// TIA Portal V20 export
FUNCTION_BLOCK "Sequence_1_StackTable"   // FB232, LAD
AUTHOR : ERsystem_FA2_DH. Kim
// stored: IsIECCheckEnabled true, MemoryReserve 100, Namespace Unit1.Em6, SetENOAutomatically false
   VAR
      statSelectedJobNumber { ExternalWritable := 'False'} : DInt;   // Evaluated Job Number
      instSequenceLADStatus { ExternalWritable := 'False'} : "LAF_StatusLadSequence";
      instSequenceLADControl { ExternalWritable := 'False'} : "LAF_ControlLadSequence";
      statTonTime { ExternalAccessible := 'False'; ExternalVisible := 'False'; ExternalWritable := 'False'} : Array[0..3999] of TON_TIME;
   END_VAR
   VAR_TEMP
      tempLoadingDone : Bool;
   END_VAR
   VAR CONSTANT
      delayTime : Time := T#300ms;
      STEP_IDLE : DInt := 1;
      STEP_IMMEDIATE_STOP : DInt := 9001;   // Step executed when an immediate stop command is triggered for the sequence (i.e. when unit is in state aborting)
      JOB_1_STEP_01 : DInt := 101;
      JOB_1_STEP_10 : DInt := 110;
      JOB_1_STEP_11 : DInt := 111;
      JOB_1_STEP_12 : DInt := 112;
      JOB_1_STEP_13 : DInt := 113;
      JOB_1_STEP_20 : DInt := 120;
      JOB_1_STEP_21 : DInt := 121;
      JOB_1_STEP_22 : DInt := 122;
      JOB_1_STEP_30 : DInt := 130;
      JOB_1_STEP_31 : DInt := 131;
      JOB_1_STEP_32 : DInt := 132;
      JOB_1_STEP_40 : DInt := 140;
      JOB_1_STEP_41 : DInt := 141;
      JOB_1_STEP_42 : DInt := 142;
      JOB_1_STEP_50 : DInt := 150;
      JOB_1_STEP_51 : DInt := 151;
      JOB_1_STEP_52 : DInt := 152;
      JOB_1_STEP_60 : DInt := 160;
      JOB_1_STEP_61 : DInt := 161;
      JOB_1_STEP_62 : DInt := 162;
      JOB_1_STEP_70 : DInt := 170;
      JOB_1_STEP_71 : DInt := 171;
      JOB_1_STEP_80 : DInt := 180;
      JOB_1_STEP_81 : DInt := 181;
      JOB_1_STEP_82 : DInt := 182;
      JOB_1_STEP_83 : DInt := 183;
      JOB_1_STEP_84 : DInt := 184;
      JOB_1_STEP_85 : DInt := 185;
      JOB_1_STEP_90 : DInt := 190;
      JOB_2_STEP_01 : DInt := 201;
      JOB_2_STEP_10 : DInt := 210;
      JOB_2_STEP_20 : DInt := 220;
      JOB_2_STEP_80 : DInt := 280;
      JOB_2_STEP_90 : DInt := 290;
      JOB_12_STEP_01 : DInt := 1201;
      JOB_12_STEP_10 : DInt := 1210;
      JOB_12_STEP_90 : DInt := 1290;
      JOB_13_STEP_01 : DInt := 1301;
      JOB_13_STEP_10 : DInt := 1310;
      JOB_13_STEP_90 : DInt := 1390;
      JOB_4_STEP_01 : DInt := 401;
      JOB_4_STEP_10 : DInt := 410;
      JOB_4_STEP_20 : DInt := 420;
      JOB_4_STEP_21 : DInt := 421;
      JOB_4_STEP_30 : DInt := 430;
      JOB_4_STEP_31 : DInt := 431;
      JOB_4_STEP_40 : DInt := 440;
      JOB_4_STEP_41 : DInt := 441;
      JOB_4_STEP_50 : DInt := 450;
      JOB_4_STEP_80 : DInt := 480;
      JOB_4_STEP_90 : DInt := 490;
      JOB_22_STEP_01 : DInt := 2201;
      JOB_22_STEP_10 : DInt := 2210;
      JOB_22_STEP_20 : DInt := 2220;
      JOB_22_STEP_21 : DInt := 2221;
      JOB_22_STEP_22 : DInt := 2222;
      JOB_22_STEP_80 : DInt := 2280;
      JOB_22_STEP_90 : DInt := 2290;
      JOB_23_STEP_01 : DInt := 2301;
      JOB_23_STEP_10 : DInt := 2310;
      JOB_23_STEP_20 : DInt := 2320;
      JOB_23_STEP_21 : DInt := 2321;
      JOB_23_STEP_22 : DInt := 2322;
      JOB_23_STEP_80 : DInt := 2380;
      JOB_23_STEP_90 : DInt := 2390;
      JOB_30_STEP_01 : DInt := 3001;
      JOB_30_STEP_10 : DInt := 3010;
      JOB_30_STEP_20 : DInt := 3020;
      JOB_30_STEP_90 : DInt := 3090;
      JOB_31_STEP_01 : DInt := 3101;
      JOB_31_STEP_10 : DInt := 3110;
      JOB_31_STEP_90 : DInt := 3190;
      FALSE : Bool := FALSE;
      TRUE : Bool := TRUE;
   END_VAR
   VAR_TEMP   // added for the SCL form of the ladder/FBD networks
      _w1 : Bool;
   END_VAR
BEGIN

REGION Network 1: BLOCK INFO HEADER
   // (company) / (C) Copyright (year)
   // ---------------------------------------------------------------------------------
   // Title:                             (Title of this block)
   // Comment/Function: (that is implemented in the block)
   // Library/Family:           (that the source is dedicated to)
   // Author:                        (department / person in charge / contact)
   // Target System:          (test system with FW version)
   // Engineering:              TIA Portal (SW version)
   // Restrictions:               (OB types, etc.)
   // Requirements:           (hardware, technological package, etc.)
   // ---------------------------------------------------------------------------------
   // Change log table:
   // Version          | Date             | Signature      | Expert in charge  | Changes applied ------------------------|----------------------|-------------------------|--------------------------------|-----------------------
   // 001.000.000 | yyyy-mm-dd | 0x00000000 | (name of expert) | First released version
END_REGION

REGION Network 2: DESCRIPTION
   // This is a template block provided by the Automation Framework. It can be used to create an own project.
   // The Block Info Header is prepared to put in your own data.
   // Description of the block could be added here and the docu created by Code2Docu.
END_REGION

REGION Network 3: ********************* CONTROL *************************
END_REGION

REGION Network 4: Sequence Control
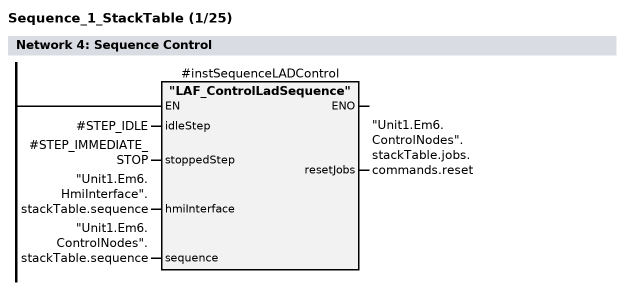
   RUNG wire#powerrail
      #instSequenceLADControl(idleStep := #STEP_IDLE, stoppedStep := #STEP_IMMEDIATE_STOP, hmiInterface := "Unit1.Em6.HmiInterface".stackTable.sequence, sequence := "Unit1.Em6.ControlNodes".stackTable.sequence, resetJobs => "Unit1.Em6.ControlNodes".stackTable.jobs.commands.reset)
   END_RUNG
   // the same network as SCL:
   #instSequenceLADControl(idleStep := #STEP_IDLE,   // "LAF_ControlLadSequence"
                           stoppedStep := #STEP_IMMEDIATE_STOP,
                           hmiInterface := "Unit1.Em6.HmiInterface".stackTable.sequence,
                           sequence := "Unit1.Em6.ControlNodes".stackTable.sequence,
                           resetJobs => "Unit1.Em6.ControlNodes".stackTable.jobs.commands.reset);
END_REGION

REGION Network 5: *************** JOB SELECT **************************
END_REGION

REGION Network 6: STEP IDLE
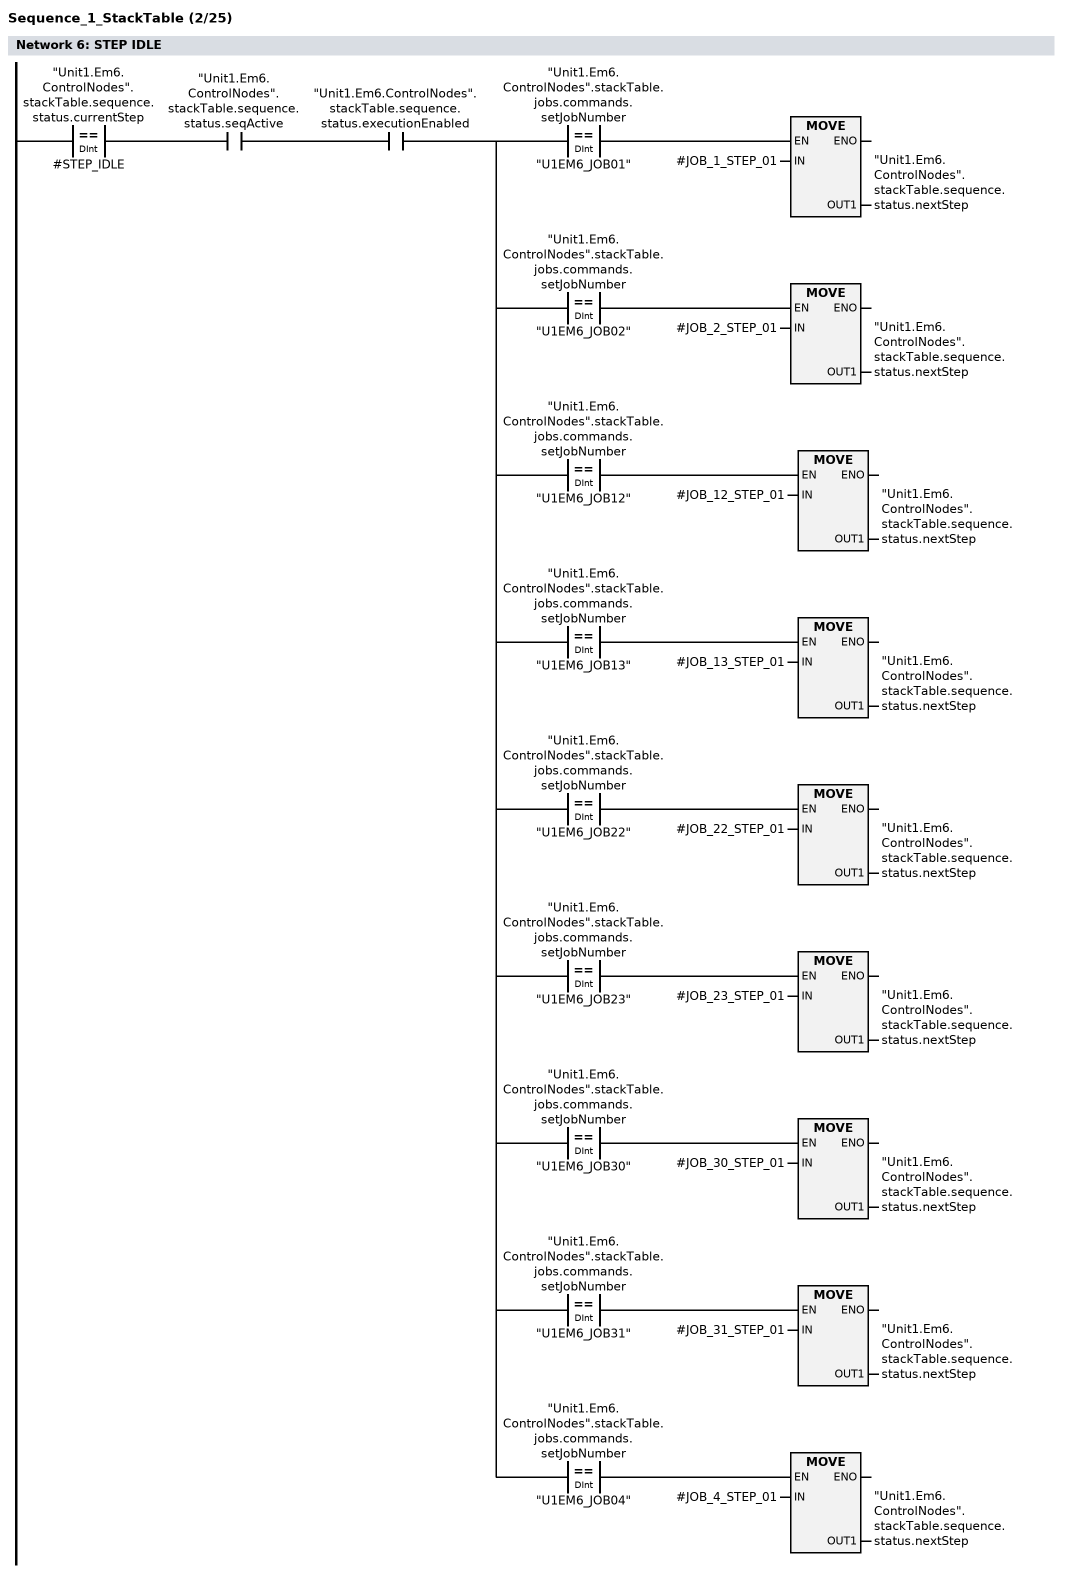
   RUNG wire#powerrail
      { S7_Templates := "SrcType := DInt" } EQ_Contact(in1 := "Unit1.Em6.ControlNodes".stackTable.sequence.status.currentStep, in2 := #STEP_IDLE)
      Contact( "Unit1.Em6.ControlNodes".stackTable.sequence.status.seqActive )
      Contact( "Unit1.Em6.ControlNodes".stackTable.sequence.status.executionEnabled )
      wire#w1
      { S7_Templates := "SrcType := DInt" } EQ_Contact(in1 := "Unit1.Em6.ControlNodes".stackTable.jobs.commands.setJobNumber, in2 := "U1EM6_JOB01")
      Move(in := #JOB_1_STEP_01, out1 => "Unit1.Em6.ControlNodes".stackTable.sequence.status.nextStep)
   END_RUNG
   RUNG wire#w1
      { S7_Templates := "SrcType := DInt" } EQ_Contact(in1 := "Unit1.Em6.ControlNodes".stackTable.jobs.commands.setJobNumber, in2 := "U1EM6_JOB02")
      Move(in := #JOB_2_STEP_01, out1 => "Unit1.Em6.ControlNodes".stackTable.sequence.status.nextStep)
   END_RUNG
   RUNG wire#w1
      { S7_Templates := "SrcType := DInt" } EQ_Contact(in1 := "Unit1.Em6.ControlNodes".stackTable.jobs.commands.setJobNumber, in2 := "U1EM6_JOB12")
      Move(in := #JOB_12_STEP_01, out1 => "Unit1.Em6.ControlNodes".stackTable.sequence.status.nextStep)
   END_RUNG
   RUNG wire#w1
      { S7_Templates := "SrcType := DInt" } EQ_Contact(in1 := "Unit1.Em6.ControlNodes".stackTable.jobs.commands.setJobNumber, in2 := "U1EM6_JOB13")
      Move(in := #JOB_13_STEP_01, out1 => "Unit1.Em6.ControlNodes".stackTable.sequence.status.nextStep)
   END_RUNG
   RUNG wire#w1
      { S7_Templates := "SrcType := DInt" } EQ_Contact(in1 := "Unit1.Em6.ControlNodes".stackTable.jobs.commands.setJobNumber, in2 := "U1EM6_JOB22")
      Move(in := #JOB_22_STEP_01, out1 => "Unit1.Em6.ControlNodes".stackTable.sequence.status.nextStep)
   END_RUNG
   RUNG wire#w1
      { S7_Templates := "SrcType := DInt" } EQ_Contact(in1 := "Unit1.Em6.ControlNodes".stackTable.jobs.commands.setJobNumber, in2 := "U1EM6_JOB23")
      Move(in := #JOB_23_STEP_01, out1 => "Unit1.Em6.ControlNodes".stackTable.sequence.status.nextStep)
   END_RUNG
   RUNG wire#w1
      { S7_Templates := "SrcType := DInt" } EQ_Contact(in1 := "Unit1.Em6.ControlNodes".stackTable.jobs.commands.setJobNumber, in2 := "U1EM6_JOB30")
      Move(in := #JOB_30_STEP_01, out1 => "Unit1.Em6.ControlNodes".stackTable.sequence.status.nextStep)
   END_RUNG
   RUNG wire#w1
      { S7_Templates := "SrcType := DInt" } EQ_Contact(in1 := "Unit1.Em6.ControlNodes".stackTable.jobs.commands.setJobNumber, in2 := "U1EM6_JOB31")
      Move(in := #JOB_31_STEP_01, out1 => "Unit1.Em6.ControlNodes".stackTable.sequence.status.nextStep)
   END_RUNG
   RUNG wire#w1
      { S7_Templates := "SrcType := DInt" } EQ_Contact(in1 := "Unit1.Em6.ControlNodes".stackTable.jobs.commands.setJobNumber, in2 := "U1EM6_JOB04")
      Move(in := #JOB_4_STEP_01, out1 => "Unit1.Em6.ControlNodes".stackTable.sequence.status.nextStep)
   END_RUNG
   // the same network as SCL:
   #_w1 := ("Unit1.Em6.ControlNodes".stackTable.sequence.status.currentStep = #STEP_IDLE) AND "Unit1.Em6.ControlNodes".stackTable.sequence.status.seqActive AND "Unit1.Em6.ControlNodes".stackTable.sequence.status.executionEnabled;
   IF #_w1 AND ("Unit1.Em6.ControlNodes".stackTable.jobs.commands.setJobNumber = "U1EM6_JOB01") THEN
       "Unit1.Em6.ControlNodes".stackTable.sequence.status.nextStep := #JOB_1_STEP_01;
   END_IF;
   IF #_w1 AND ("Unit1.Em6.ControlNodes".stackTable.jobs.commands.setJobNumber = "U1EM6_JOB02") THEN
       "Unit1.Em6.ControlNodes".stackTable.sequence.status.nextStep := #JOB_2_STEP_01;
   END_IF;
   IF #_w1 AND ("Unit1.Em6.ControlNodes".stackTable.jobs.commands.setJobNumber = "U1EM6_JOB12") THEN
       "Unit1.Em6.ControlNodes".stackTable.sequence.status.nextStep := #JOB_12_STEP_01;
   END_IF;
   IF #_w1 AND ("Unit1.Em6.ControlNodes".stackTable.jobs.commands.setJobNumber = "U1EM6_JOB13") THEN
       "Unit1.Em6.ControlNodes".stackTable.sequence.status.nextStep := #JOB_13_STEP_01;
   END_IF;
   IF #_w1 AND ("Unit1.Em6.ControlNodes".stackTable.jobs.commands.setJobNumber = "U1EM6_JOB22") THEN
       "Unit1.Em6.ControlNodes".stackTable.sequence.status.nextStep := #JOB_22_STEP_01;
   END_IF;
   IF #_w1 AND ("Unit1.Em6.ControlNodes".stackTable.jobs.commands.setJobNumber = "U1EM6_JOB23") THEN
       "Unit1.Em6.ControlNodes".stackTable.sequence.status.nextStep := #JOB_23_STEP_01;
   END_IF;
   IF #_w1 AND ("Unit1.Em6.ControlNodes".stackTable.jobs.commands.setJobNumber = "U1EM6_JOB30") THEN
       "Unit1.Em6.ControlNodes".stackTable.sequence.status.nextStep := #JOB_30_STEP_01;
   END_IF;
   IF #_w1 AND ("Unit1.Em6.ControlNodes".stackTable.jobs.commands.setJobNumber = "U1EM6_JOB31") THEN
       "Unit1.Em6.ControlNodes".stackTable.sequence.status.nextStep := #JOB_31_STEP_01;
   END_IF;
   IF #_w1 AND ("Unit1.Em6.ControlNodes".stackTable.jobs.commands.setJobNumber = "U1EM6_JOB04") THEN
       "Unit1.Em6.ControlNodes".stackTable.sequence.status.nextStep := #JOB_4_STEP_01;
   END_IF;
END_REGION

REGION Network 7: *************** JOB[1] EM HOMING ************************
END_REGION

REGION Network 8: Step[101] : JOB[1] Condition
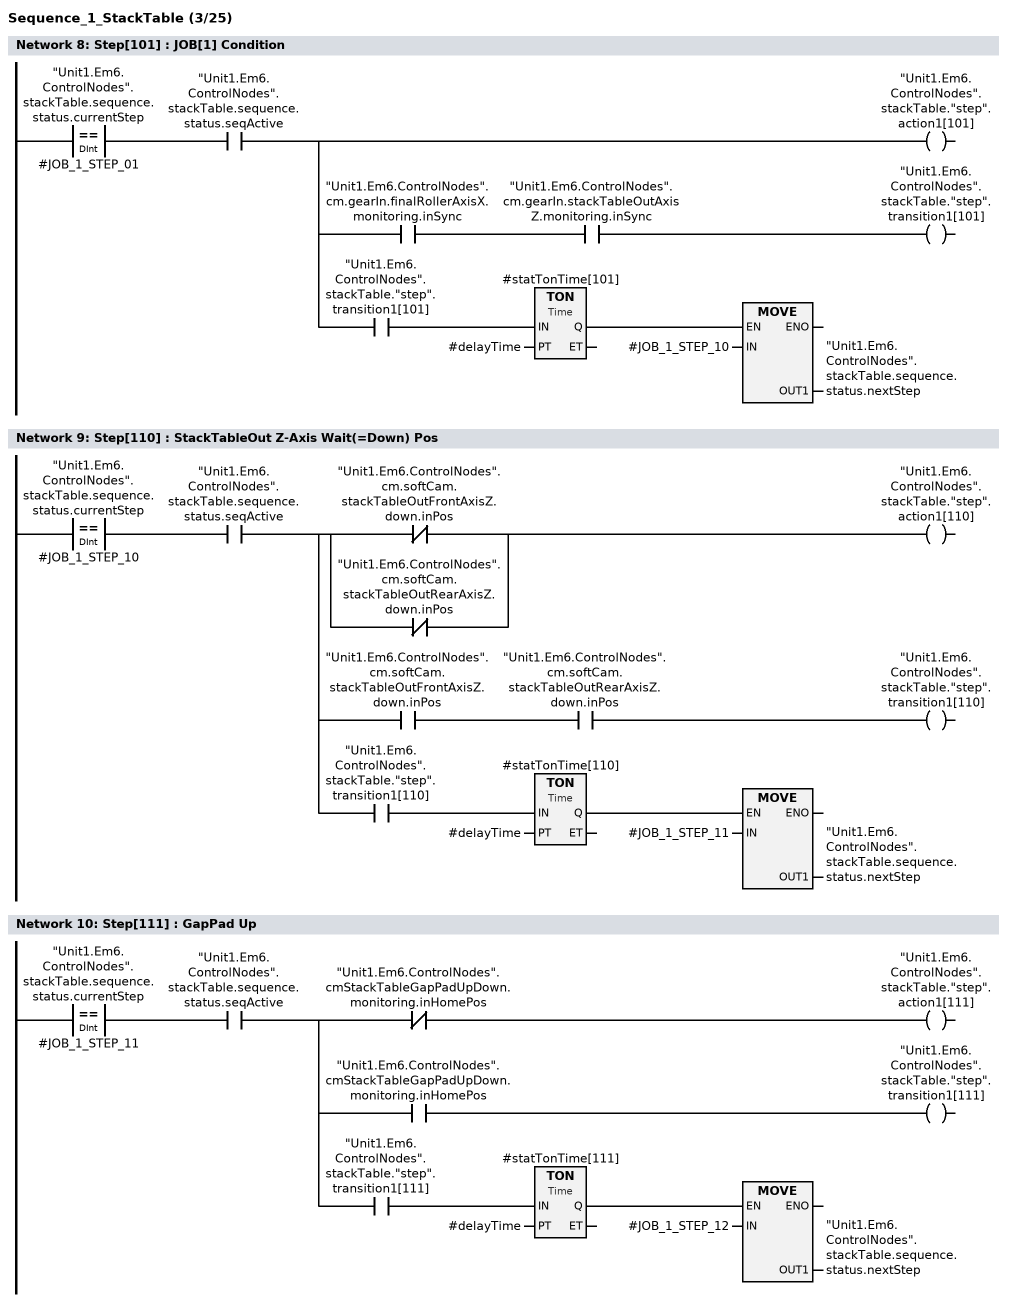
   RUNG wire#powerrail
      { S7_Templates := "SrcType := DInt" } EQ_Contact(in1 := "Unit1.Em6.ControlNodes".stackTable.sequence.status.currentStep, in2 := #JOB_1_STEP_01)
      Contact( "Unit1.Em6.ControlNodes".stackTable.sequence.status.seqActive )
      wire#w1
      Coil( "Unit1.Em6.ControlNodes".stackTable."step".action1[101] )
   END_RUNG
   RUNG wire#w1
      Contact( "Unit1.Em6.ControlNodes".cm.gearIn.finalRollerAxisX.monitoring.inSync )
      Contact( "Unit1.Em6.ControlNodes".cm.gearIn.stackTableOutAxisZ.monitoring.inSync )
      Coil( "Unit1.Em6.ControlNodes".stackTable."step".transition1[101] )
   END_RUNG
   RUNG wire#w1
      Contact( "Unit1.Em6.ControlNodes".stackTable."step".transition1[101] )
      { S7_Templates := "time_type := Time" } #statTonTime[101].TON(pt := #delayTime, et =>)
      Move(in := #JOB_1_STEP_10, out1 => "Unit1.Em6.ControlNodes".stackTable.sequence.status.nextStep)
   END_RUNG
   // the same network as SCL:
   "Unit1.Em6.ControlNodes".stackTable."step".action1[101] := ("Unit1.Em6.ControlNodes".stackTable.sequence.status.currentStep = #JOB_1_STEP_01) AND "Unit1.Em6.ControlNodes".stackTable.sequence.status.seqActive;
   "Unit1.Em6.ControlNodes".stackTable."step".transition1[101] := ("Unit1.Em6.ControlNodes".stackTable.sequence.status.currentStep = #JOB_1_STEP_01) AND "Unit1.Em6.ControlNodes".stackTable.sequence.status.seqActive AND "Unit1.Em6.ControlNodes".cm.gearIn.finalRollerAxisX.monitoring.inSync AND "Unit1.Em6.ControlNodes".cm.gearIn.stackTableOutAxisZ.monitoring.inSync;
   #statTonTime[101].TON(IN := ("Unit1.Em6.ControlNodes".stackTable.sequence.status.currentStep = #JOB_1_STEP_01) AND "Unit1.Em6.ControlNodes".stackTable.sequence.status.seqActive AND "Unit1.Em6.ControlNodes".stackTable."step".transition1[101],
                         PT := #delayTime);
   IF #statTonTime[101].Q THEN
       "Unit1.Em6.ControlNodes".stackTable.sequence.status.nextStep := #JOB_1_STEP_10;
   END_IF;
END_REGION

REGION Network 9: Step[110] : StackTableOut Z-Axis Wait(=Down) Pos
   RUNG wire#powerrail
      { S7_Templates := "SrcType := DInt" } EQ_Contact(in1 := "Unit1.Em6.ControlNodes".stackTable.sequence.status.currentStep, in2 := #JOB_1_STEP_10)
      Contact( "Unit1.Em6.ControlNodes".stackTable.sequence.status.seqActive )
      wire#w1
      I_Contact( "Unit1.Em6.ControlNodes".cm.softCam.stackTableOutFrontAxisZ.down.inPos )
      wire#w2
      Coil( "Unit1.Em6.ControlNodes".stackTable."step".action1[110] )
   END_RUNG
   RUNG wire#w1
      I_Contact( "Unit1.Em6.ControlNodes".cm.softCam.stackTableOutRearAxisZ.down.inPos )
   END_RUNG wire#w2
   RUNG wire#w1
      Contact( "Unit1.Em6.ControlNodes".cm.softCam.stackTableOutFrontAxisZ.down.inPos )
      Contact( "Unit1.Em6.ControlNodes".cm.softCam.stackTableOutRearAxisZ.down.inPos )
      Coil( "Unit1.Em6.ControlNodes".stackTable."step".transition1[110] )
   END_RUNG
   RUNG wire#w1
      Contact( "Unit1.Em6.ControlNodes".stackTable."step".transition1[110] )
      { S7_Templates := "time_type := Time" } #statTonTime[110].TON(pt := #delayTime, et =>)
      Move(in := #JOB_1_STEP_11, out1 => "Unit1.Em6.ControlNodes".stackTable.sequence.status.nextStep)
   END_RUNG
   // the same network as SCL:
   #_w1 := ("Unit1.Em6.ControlNodes".stackTable.sequence.status.currentStep = #JOB_1_STEP_10) AND "Unit1.Em6.ControlNodes".stackTable.sequence.status.seqActive;
   "Unit1.Em6.ControlNodes".stackTable."step".action1[110] := #_w1 AND (NOT "Unit1.Em6.ControlNodes".cm.softCam.stackTableOutFrontAxisZ.down.inPos OR NOT "Unit1.Em6.ControlNodes".cm.softCam.stackTableOutRearAxisZ.down.inPos);
   "Unit1.Em6.ControlNodes".stackTable."step".transition1[110] := #_w1 AND "Unit1.Em6.ControlNodes".cm.softCam.stackTableOutFrontAxisZ.down.inPos AND "Unit1.Em6.ControlNodes".cm.softCam.stackTableOutRearAxisZ.down.inPos;
   #statTonTime[110].TON(IN := #_w1 AND "Unit1.Em6.ControlNodes".stackTable."step".transition1[110],
                         PT := #delayTime);
   IF #statTonTime[110].Q THEN
       "Unit1.Em6.ControlNodes".stackTable.sequence.status.nextStep := #JOB_1_STEP_11;
   END_IF;
END_REGION

REGION Network 10: Step[111] : GapPad Up
   RUNG wire#powerrail
      { S7_Templates := "SrcType := DInt" } EQ_Contact(in1 := "Unit1.Em6.ControlNodes".stackTable.sequence.status.currentStep, in2 := #JOB_1_STEP_11)
      Contact( "Unit1.Em6.ControlNodes".stackTable.sequence.status.seqActive )
      wire#w1
      I_Contact( "Unit1.Em6.ControlNodes".cmStackTableGapPadUpDown.monitoring.inHomePos )
      Coil( "Unit1.Em6.ControlNodes".stackTable."step".action1[111] )
   END_RUNG
   RUNG wire#w1
      Contact( "Unit1.Em6.ControlNodes".cmStackTableGapPadUpDown.monitoring.inHomePos )
      Coil( "Unit1.Em6.ControlNodes".stackTable."step".transition1[111] )
   END_RUNG
   RUNG wire#w1
      Contact( "Unit1.Em6.ControlNodes".stackTable."step".transition1[111] )
      { S7_Templates := "time_type := Time" } #statTonTime[111].TON(pt := #delayTime, et =>)
      Move(in := #JOB_1_STEP_12, out1 => "Unit1.Em6.ControlNodes".stackTable.sequence.status.nextStep)
   END_RUNG
   // the same network as SCL:
   #_w1 := ("Unit1.Em6.ControlNodes".stackTable.sequence.status.currentStep = #JOB_1_STEP_11) AND "Unit1.Em6.ControlNodes".stackTable.sequence.status.seqActive;
   "Unit1.Em6.ControlNodes".stackTable."step".action1[111] := #_w1 AND NOT "Unit1.Em6.ControlNodes".cmStackTableGapPadUpDown.monitoring.inHomePos;
   "Unit1.Em6.ControlNodes".stackTable."step".transition1[111] := #_w1 AND "Unit1.Em6.ControlNodes".cmStackTableGapPadUpDown.monitoring.inHomePos;
   #statTonTime[111].TON(IN := #_w1 AND "Unit1.Em6.ControlNodes".stackTable."step".transition1[111],
                         PT := #delayTime);
   IF #statTonTime[111].Q THEN
       "Unit1.Em6.ControlNodes".stackTable.sequence.status.nextStep := #JOB_1_STEP_12;
   END_IF;
END_REGION

REGION Network 11: Step[112] : A,C.Mendrel Clamp Work Pos
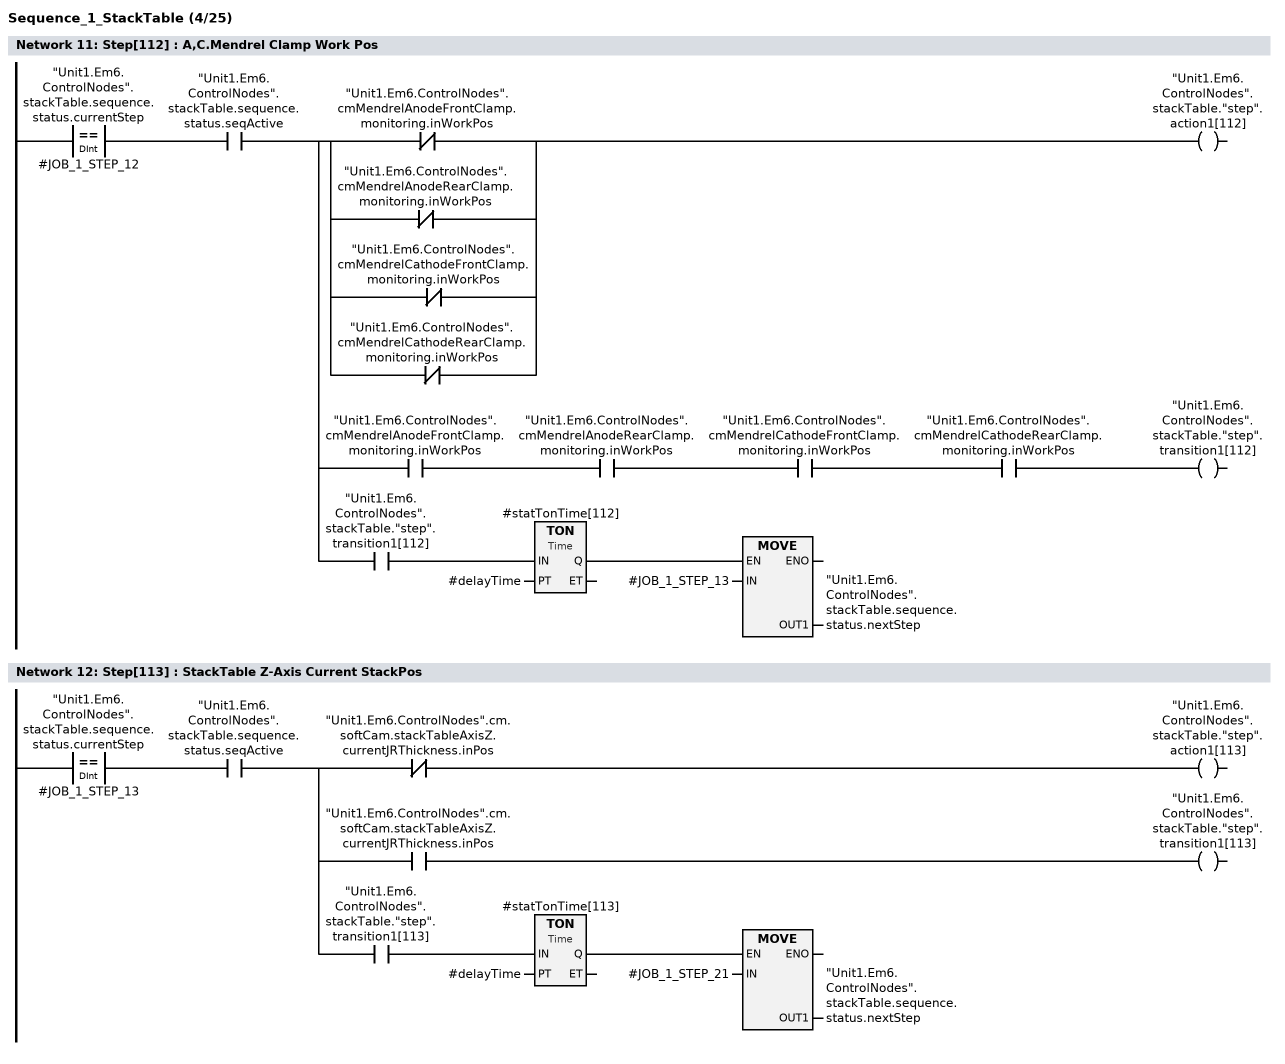
   RUNG wire#powerrail
      { S7_Templates := "SrcType := DInt" } EQ_Contact(in1 := "Unit1.Em6.ControlNodes".stackTable.sequence.status.currentStep, in2 := #JOB_1_STEP_12)
      Contact( "Unit1.Em6.ControlNodes".stackTable.sequence.status.seqActive )
      wire#w1
      I_Contact( "Unit1.Em6.ControlNodes".cmMendrelAnodeFrontClamp.monitoring.inWorkPos )
      wire#w2
      Coil( "Unit1.Em6.ControlNodes".stackTable."step".action1[112] )
   END_RUNG
   RUNG wire#w1
      I_Contact( "Unit1.Em6.ControlNodes".cmMendrelAnodeRearClamp.monitoring.inWorkPos )
   END_RUNG wire#w2
   RUNG wire#w1
      I_Contact( "Unit1.Em6.ControlNodes".cmMendrelCathodeFrontClamp.monitoring.inWorkPos )
   END_RUNG wire#w2
   RUNG wire#w1
      I_Contact( "Unit1.Em6.ControlNodes".cmMendrelCathodeRearClamp.monitoring.inWorkPos )
   END_RUNG wire#w2
   RUNG wire#w1
      Contact( "Unit1.Em6.ControlNodes".cmMendrelAnodeFrontClamp.monitoring.inWorkPos )
      Contact( "Unit1.Em6.ControlNodes".cmMendrelAnodeRearClamp.monitoring.inWorkPos )
      Contact( "Unit1.Em6.ControlNodes".cmMendrelCathodeFrontClamp.monitoring.inWorkPos )
      Contact( "Unit1.Em6.ControlNodes".cmMendrelCathodeRearClamp.monitoring.inWorkPos )
      Coil( "Unit1.Em6.ControlNodes".stackTable."step".transition1[112] )
   END_RUNG
   RUNG wire#w1
      Contact( "Unit1.Em6.ControlNodes".stackTable."step".transition1[112] )
      { S7_Templates := "time_type := Time" } #statTonTime[112].TON(pt := #delayTime, et =>)
      Move(in := #JOB_1_STEP_13, out1 => "Unit1.Em6.ControlNodes".stackTable.sequence.status.nextStep)
   END_RUNG
   // the same network as SCL:
   #_w1 := ("Unit1.Em6.ControlNodes".stackTable.sequence.status.currentStep = #JOB_1_STEP_12) AND "Unit1.Em6.ControlNodes".stackTable.sequence.status.seqActive;
   "Unit1.Em6.ControlNodes".stackTable."step".action1[112] := #_w1 AND (NOT "Unit1.Em6.ControlNodes".cmMendrelAnodeFrontClamp.monitoring.inWorkPos OR NOT "Unit1.Em6.ControlNodes".cmMendrelAnodeRearClamp.monitoring.inWorkPos OR NOT "Unit1.Em6.ControlNodes".cmMendrelCathodeFrontClamp.monitoring.inWorkPos OR NOT "Unit1.Em6.ControlNodes".cmMendrelCathodeRearClamp.monitoring.inWorkPos);
   "Unit1.Em6.ControlNodes".stackTable."step".transition1[112] := #_w1 AND "Unit1.Em6.ControlNodes".cmMendrelAnodeFrontClamp.monitoring.inWorkPos AND "Unit1.Em6.ControlNodes".cmMendrelAnodeRearClamp.monitoring.inWorkPos AND "Unit1.Em6.ControlNodes".cmMendrelCathodeFrontClamp.monitoring.inWorkPos AND "Unit1.Em6.ControlNodes".cmMendrelCathodeRearClamp.monitoring.inWorkPos;
   #statTonTime[112].TON(IN := #_w1 AND "Unit1.Em6.ControlNodes".stackTable."step".transition1[112],
                         PT := #delayTime);
   IF #statTonTime[112].Q THEN
       "Unit1.Em6.ControlNodes".stackTable.sequence.status.nextStep := #JOB_1_STEP_13;
   END_IF;
END_REGION

REGION Network 12: Step[113] : StackTable Z-Axis Current StackPos
   RUNG wire#powerrail
      { S7_Templates := "SrcType := DInt" } EQ_Contact(in1 := "Unit1.Em6.ControlNodes".stackTable.sequence.status.currentStep, in2 := #JOB_1_STEP_13)
      Contact( "Unit1.Em6.ControlNodes".stackTable.sequence.status.seqActive )
      wire#w1
      I_Contact( "Unit1.Em6.ControlNodes".cm.softCam.stackTableAxisZ.currentJRThickness.inPos )
      Coil( "Unit1.Em6.ControlNodes".stackTable."step".action1[113] )
   END_RUNG
   RUNG wire#w1
      Contact( "Unit1.Em6.ControlNodes".cm.softCam.stackTableAxisZ.currentJRThickness.inPos )
      Coil( "Unit1.Em6.ControlNodes".stackTable."step".transition1[113] )
   END_RUNG
   RUNG wire#w1
      Contact( "Unit1.Em6.ControlNodes".stackTable."step".transition1[113] )
      { S7_Templates := "time_type := Time" } #statTonTime[113].TON(pt := #delayTime, et =>)
      Move(in := #JOB_1_STEP_21, out1 => "Unit1.Em6.ControlNodes".stackTable.sequence.status.nextStep)
   END_RUNG
   // the same network as SCL:
   #_w1 := ("Unit1.Em6.ControlNodes".stackTable.sequence.status.currentStep = #JOB_1_STEP_13) AND "Unit1.Em6.ControlNodes".stackTable.sequence.status.seqActive;
   "Unit1.Em6.ControlNodes".stackTable."step".action1[113] := #_w1 AND NOT "Unit1.Em6.ControlNodes".cm.softCam.stackTableAxisZ.currentJRThickness.inPos;
   "Unit1.Em6.ControlNodes".stackTable."step".transition1[113] := #_w1 AND "Unit1.Em6.ControlNodes".cm.softCam.stackTableAxisZ.currentJRThickness.inPos;
   #statTonTime[113].TON(IN := #_w1 AND "Unit1.Em6.ControlNodes".stackTable."step".transition1[113],
                         PT := #delayTime);
   IF #statTonTime[113].Q THEN
       "Unit1.Em6.ControlNodes".stackTable.sequence.status.nextStep := #JOB_1_STEP_21;
   END_IF;
END_REGION

REGION Network 14: Step[121] : C.Mendrel Y,Z-Axis Work Pos
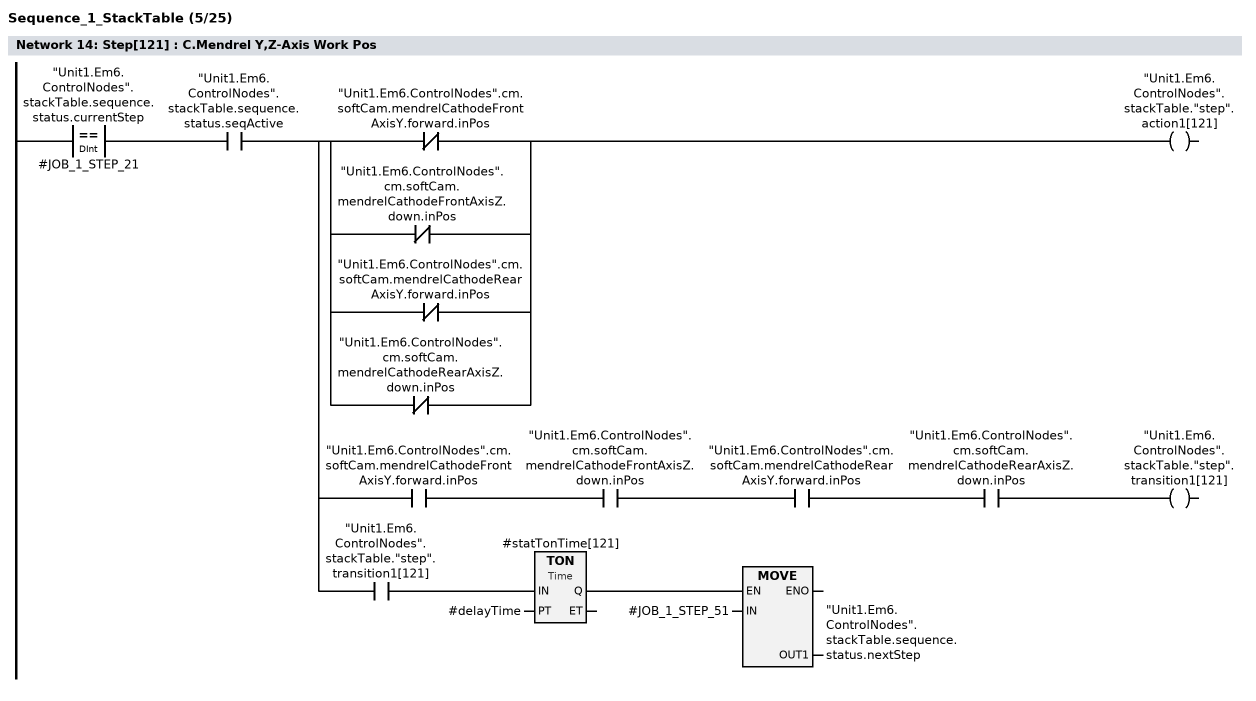
   RUNG wire#powerrail
      { S7_Templates := "SrcType := DInt" } EQ_Contact(in1 := "Unit1.Em6.ControlNodes".stackTable.sequence.status.currentStep, in2 := #JOB_1_STEP_21)
      Contact( "Unit1.Em6.ControlNodes".stackTable.sequence.status.seqActive )
      wire#w1
      I_Contact( "Unit1.Em6.ControlNodes".cm.softCam.mendrelCathodeFrontAxisY.forward.inPos )
      wire#w2
      Coil( "Unit1.Em6.ControlNodes".stackTable."step".action1[121] )
   END_RUNG
   RUNG wire#w1
      I_Contact( "Unit1.Em6.ControlNodes".cm.softCam.mendrelCathodeFrontAxisZ.down.inPos )
   END_RUNG wire#w2
   RUNG wire#w1
      I_Contact( "Unit1.Em6.ControlNodes".cm.softCam.mendrelCathodeRearAxisY.forward.inPos )
   END_RUNG wire#w2
   RUNG wire#w1
      I_Contact( "Unit1.Em6.ControlNodes".cm.softCam.mendrelCathodeRearAxisZ.down.inPos )
   END_RUNG wire#w2
   RUNG wire#w1
      Contact( "Unit1.Em6.ControlNodes".cm.softCam.mendrelCathodeFrontAxisY.forward.inPos )
      Contact( "Unit1.Em6.ControlNodes".cm.softCam.mendrelCathodeFrontAxisZ.down.inPos )
      Contact( "Unit1.Em6.ControlNodes".cm.softCam.mendrelCathodeRearAxisY.forward.inPos )
      Contact( "Unit1.Em6.ControlNodes".cm.softCam.mendrelCathodeRearAxisZ.down.inPos )
      Coil( "Unit1.Em6.ControlNodes".stackTable."step".transition1[121] )
   END_RUNG
   RUNG wire#w1
      Contact( "Unit1.Em6.ControlNodes".stackTable."step".transition1[121] )
      { S7_Templates := "time_type := Time" } #statTonTime[121].TON(pt := #delayTime, et =>)
      Move(in := #JOB_1_STEP_51, out1 => "Unit1.Em6.ControlNodes".stackTable.sequence.status.nextStep)
   END_RUNG
   // the same network as SCL:
   #_w1 := ("Unit1.Em6.ControlNodes".stackTable.sequence.status.currentStep = #JOB_1_STEP_21) AND "Unit1.Em6.ControlNodes".stackTable.sequence.status.seqActive;
   "Unit1.Em6.ControlNodes".stackTable."step".action1[121] := #_w1 AND (NOT "Unit1.Em6.ControlNodes".cm.softCam.mendrelCathodeFrontAxisY.forward.inPos OR NOT "Unit1.Em6.ControlNodes".cm.softCam.mendrelCathodeFrontAxisZ.down.inPos OR NOT "Unit1.Em6.ControlNodes".cm.softCam.mendrelCathodeRearAxisY.forward.inPos OR NOT "Unit1.Em6.ControlNodes".cm.softCam.mendrelCathodeRearAxisZ.down.inPos);
   "Unit1.Em6.ControlNodes".stackTable."step".transition1[121] := #_w1 AND "Unit1.Em6.ControlNodes".cm.softCam.mendrelCathodeFrontAxisY.forward.inPos AND "Unit1.Em6.ControlNodes".cm.softCam.mendrelCathodeFrontAxisZ.down.inPos AND "Unit1.Em6.ControlNodes".cm.softCam.mendrelCathodeRearAxisY.forward.inPos AND "Unit1.Em6.ControlNodes".cm.softCam.mendrelCathodeRearAxisZ.down.inPos;
   #statTonTime[121].TON(IN := #_w1 AND "Unit1.Em6.ControlNodes".stackTable."step".transition1[121],
                         PT := #delayTime);
   IF #statTonTime[121].Q THEN
       "Unit1.Em6.ControlNodes".stackTable.sequence.status.nextStep := #JOB_1_STEP_51;
   END_IF;
END_REGION

REGION Network 15: Step[151] : A.Mendrel Y,Z-Axis Work Pos
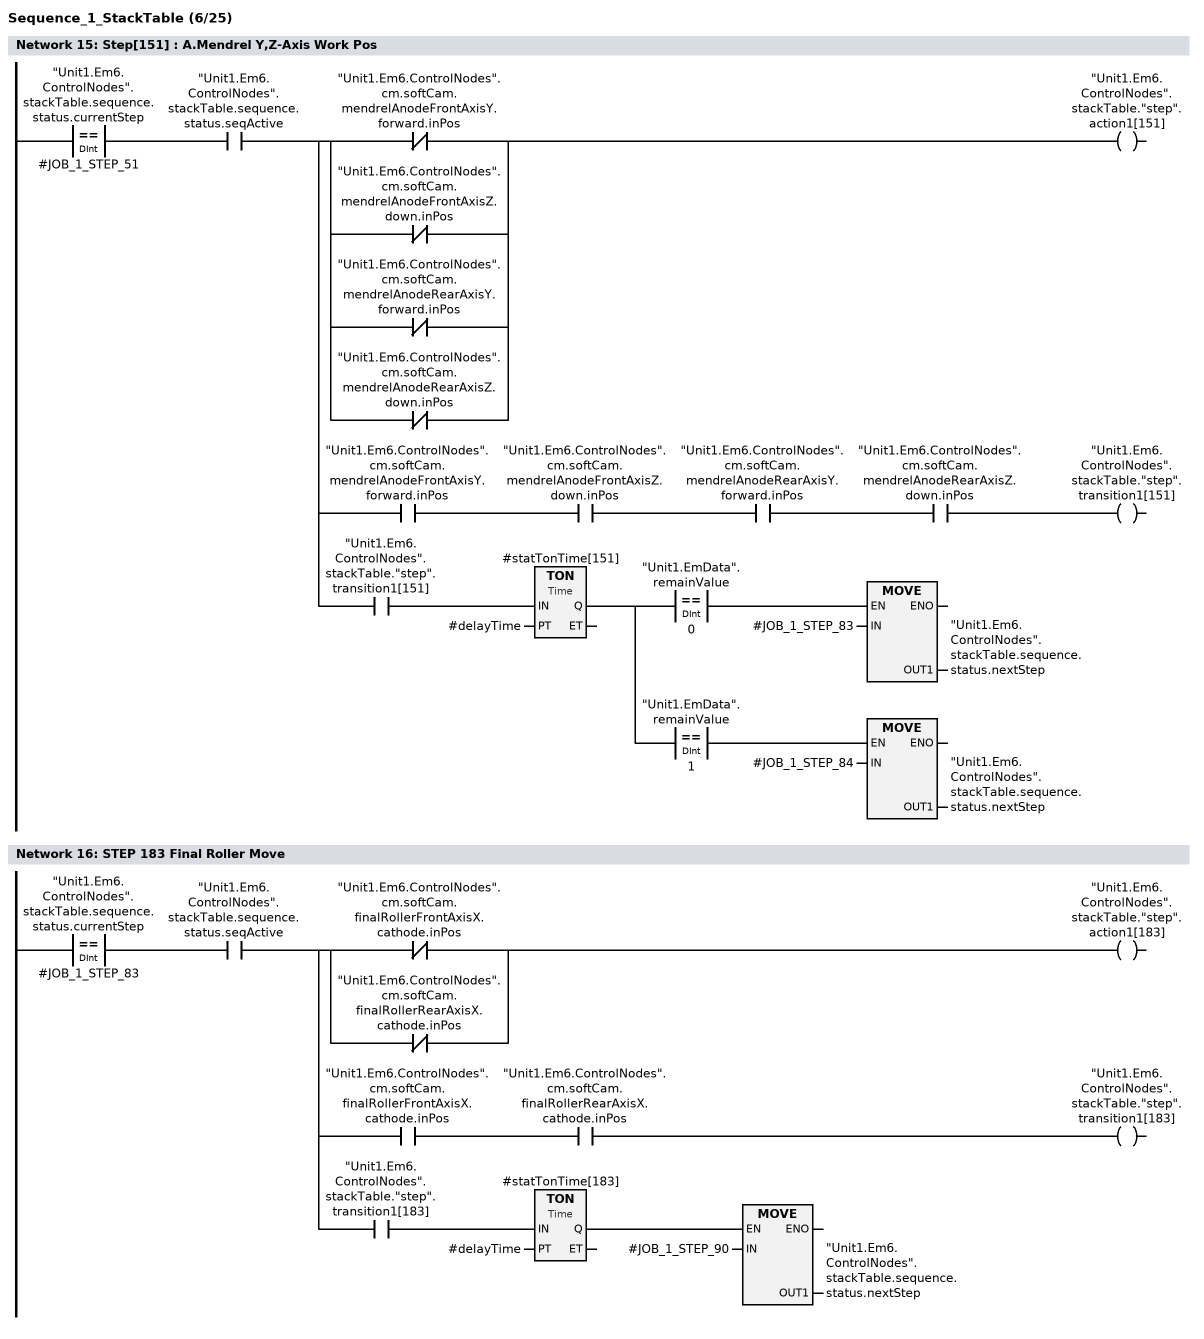
   RUNG wire#powerrail
      { S7_Templates := "SrcType := DInt" } EQ_Contact(in1 := "Unit1.Em6.ControlNodes".stackTable.sequence.status.currentStep, in2 := #JOB_1_STEP_51)
      Contact( "Unit1.Em6.ControlNodes".stackTable.sequence.status.seqActive )
      wire#w1
      I_Contact( "Unit1.Em6.ControlNodes".cm.softCam.mendrelAnodeFrontAxisY.forward.inPos )
      wire#w2
      Coil( "Unit1.Em6.ControlNodes".stackTable."step".action1[151] )
   END_RUNG
   RUNG wire#w1
      I_Contact( "Unit1.Em6.ControlNodes".cm.softCam.mendrelAnodeFrontAxisZ.down.inPos )
   END_RUNG wire#w2
   RUNG wire#w1
      I_Contact( "Unit1.Em6.ControlNodes".cm.softCam.mendrelAnodeRearAxisY.forward.inPos )
   END_RUNG wire#w2
   RUNG wire#w1
      I_Contact( "Unit1.Em6.ControlNodes".cm.softCam.mendrelAnodeRearAxisZ.down.inPos )
   END_RUNG wire#w2
   RUNG wire#w1
      Contact( "Unit1.Em6.ControlNodes".cm.softCam.mendrelAnodeFrontAxisY.forward.inPos )
      Contact( "Unit1.Em6.ControlNodes".cm.softCam.mendrelAnodeFrontAxisZ.down.inPos )
      Contact( "Unit1.Em6.ControlNodes".cm.softCam.mendrelAnodeRearAxisY.forward.inPos )
      Contact( "Unit1.Em6.ControlNodes".cm.softCam.mendrelAnodeRearAxisZ.down.inPos )
      Coil( "Unit1.Em6.ControlNodes".stackTable."step".transition1[151] )
   END_RUNG
   RUNG wire#w1
      Contact( "Unit1.Em6.ControlNodes".stackTable."step".transition1[151] )
      { S7_Templates := "time_type := Time" } #statTonTime[151].TON(pt := #delayTime, et =>)
      wire#w3
      { S7_Templates := "SrcType := DInt" } EQ_Contact(in1 := "Unit1.EmData".remainValue, in2 := 0)
      Move(in := #JOB_1_STEP_83, out1 => "Unit1.Em6.ControlNodes".stackTable.sequence.status.nextStep)
   END_RUNG
   RUNG wire#w3
      { S7_Templates := "SrcType := DInt" } EQ_Contact(in1 := "Unit1.EmData".remainValue, in2 := 1)
      Move(in := #JOB_1_STEP_84, out1 => "Unit1.Em6.ControlNodes".stackTable.sequence.status.nextStep)
   END_RUNG
   // the same network as SCL:
   #_w1 := ("Unit1.Em6.ControlNodes".stackTable.sequence.status.currentStep = #JOB_1_STEP_51) AND "Unit1.Em6.ControlNodes".stackTable.sequence.status.seqActive;
   "Unit1.Em6.ControlNodes".stackTable."step".action1[151] := #_w1 AND (NOT "Unit1.Em6.ControlNodes".cm.softCam.mendrelAnodeFrontAxisY.forward.inPos OR NOT "Unit1.Em6.ControlNodes".cm.softCam.mendrelAnodeFrontAxisZ.down.inPos OR NOT "Unit1.Em6.ControlNodes".cm.softCam.mendrelAnodeRearAxisY.forward.inPos OR NOT "Unit1.Em6.ControlNodes".cm.softCam.mendrelAnodeRearAxisZ.down.inPos);
   "Unit1.Em6.ControlNodes".stackTable."step".transition1[151] := #_w1 AND "Unit1.Em6.ControlNodes".cm.softCam.mendrelAnodeFrontAxisY.forward.inPos AND "Unit1.Em6.ControlNodes".cm.softCam.mendrelAnodeFrontAxisZ.down.inPos AND "Unit1.Em6.ControlNodes".cm.softCam.mendrelAnodeRearAxisY.forward.inPos AND "Unit1.Em6.ControlNodes".cm.softCam.mendrelAnodeRearAxisZ.down.inPos;
   #statTonTime[151].TON(IN := #_w1 AND "Unit1.Em6.ControlNodes".stackTable."step".transition1[151],
                         PT := #delayTime);
   IF #statTonTime[151].Q AND ("Unit1.EmData".remainValue = 0) THEN
       "Unit1.Em6.ControlNodes".stackTable.sequence.status.nextStep := #JOB_1_STEP_83;
   END_IF;
   IF #statTonTime[151].Q AND ("Unit1.EmData".remainValue = 1) THEN
       "Unit1.Em6.ControlNodes".stackTable.sequence.status.nextStep := #JOB_1_STEP_84;
   END_IF;
END_REGION

REGION Network 16: STEP 183 Final Roller Move
   RUNG wire#powerrail
      { S7_Templates := "SrcType := DInt" } EQ_Contact(in1 := "Unit1.Em6.ControlNodes".stackTable.sequence.status.currentStep, in2 := #JOB_1_STEP_83)
      Contact( "Unit1.Em6.ControlNodes".stackTable.sequence.status.seqActive )
      wire#w1
      I_Contact( "Unit1.Em6.ControlNodes".cm.softCam.finalRollerFrontAxisX.cathode.inPos )
      wire#w2
      Coil( "Unit1.Em6.ControlNodes".stackTable."step".action1[183] )
   END_RUNG
   RUNG wire#w1
      I_Contact( "Unit1.Em6.ControlNodes".cm.softCam.finalRollerRearAxisX.cathode.inPos )
   END_RUNG wire#w2
   RUNG wire#w1
      Contact( "Unit1.Em6.ControlNodes".cm.softCam.finalRollerFrontAxisX.cathode.inPos )
      Contact( "Unit1.Em6.ControlNodes".cm.softCam.finalRollerRearAxisX.cathode.inPos )
      Coil( "Unit1.Em6.ControlNodes".stackTable."step".transition1[183] )
   END_RUNG
   RUNG wire#w1
      Contact( "Unit1.Em6.ControlNodes".stackTable."step".transition1[183] )
      { S7_Templates := "time_type := Time" } #statTonTime[183].TON(pt := #delayTime, et =>)
      Move(in := #JOB_1_STEP_90, out1 => "Unit1.Em6.ControlNodes".stackTable.sequence.status.nextStep)
   END_RUNG
   // the same network as SCL:
   #_w1 := ("Unit1.Em6.ControlNodes".stackTable.sequence.status.currentStep = #JOB_1_STEP_83) AND "Unit1.Em6.ControlNodes".stackTable.sequence.status.seqActive;
   "Unit1.Em6.ControlNodes".stackTable."step".action1[183] := #_w1 AND (NOT "Unit1.Em6.ControlNodes".cm.softCam.finalRollerFrontAxisX.cathode.inPos OR NOT "Unit1.Em6.ControlNodes".cm.softCam.finalRollerRearAxisX.cathode.inPos);
   "Unit1.Em6.ControlNodes".stackTable."step".transition1[183] := #_w1 AND "Unit1.Em6.ControlNodes".cm.softCam.finalRollerFrontAxisX.cathode.inPos AND "Unit1.Em6.ControlNodes".cm.softCam.finalRollerRearAxisX.cathode.inPos;
   #statTonTime[183].TON(IN := #_w1 AND "Unit1.Em6.ControlNodes".stackTable."step".transition1[183],
                         PT := #delayTime);
   IF #statTonTime[183].Q THEN
       "Unit1.Em6.ControlNodes".stackTable.sequence.status.nextStep := #JOB_1_STEP_90;
   END_IF;
END_REGION

REGION Network 17: STEP 184 Final Roller Move
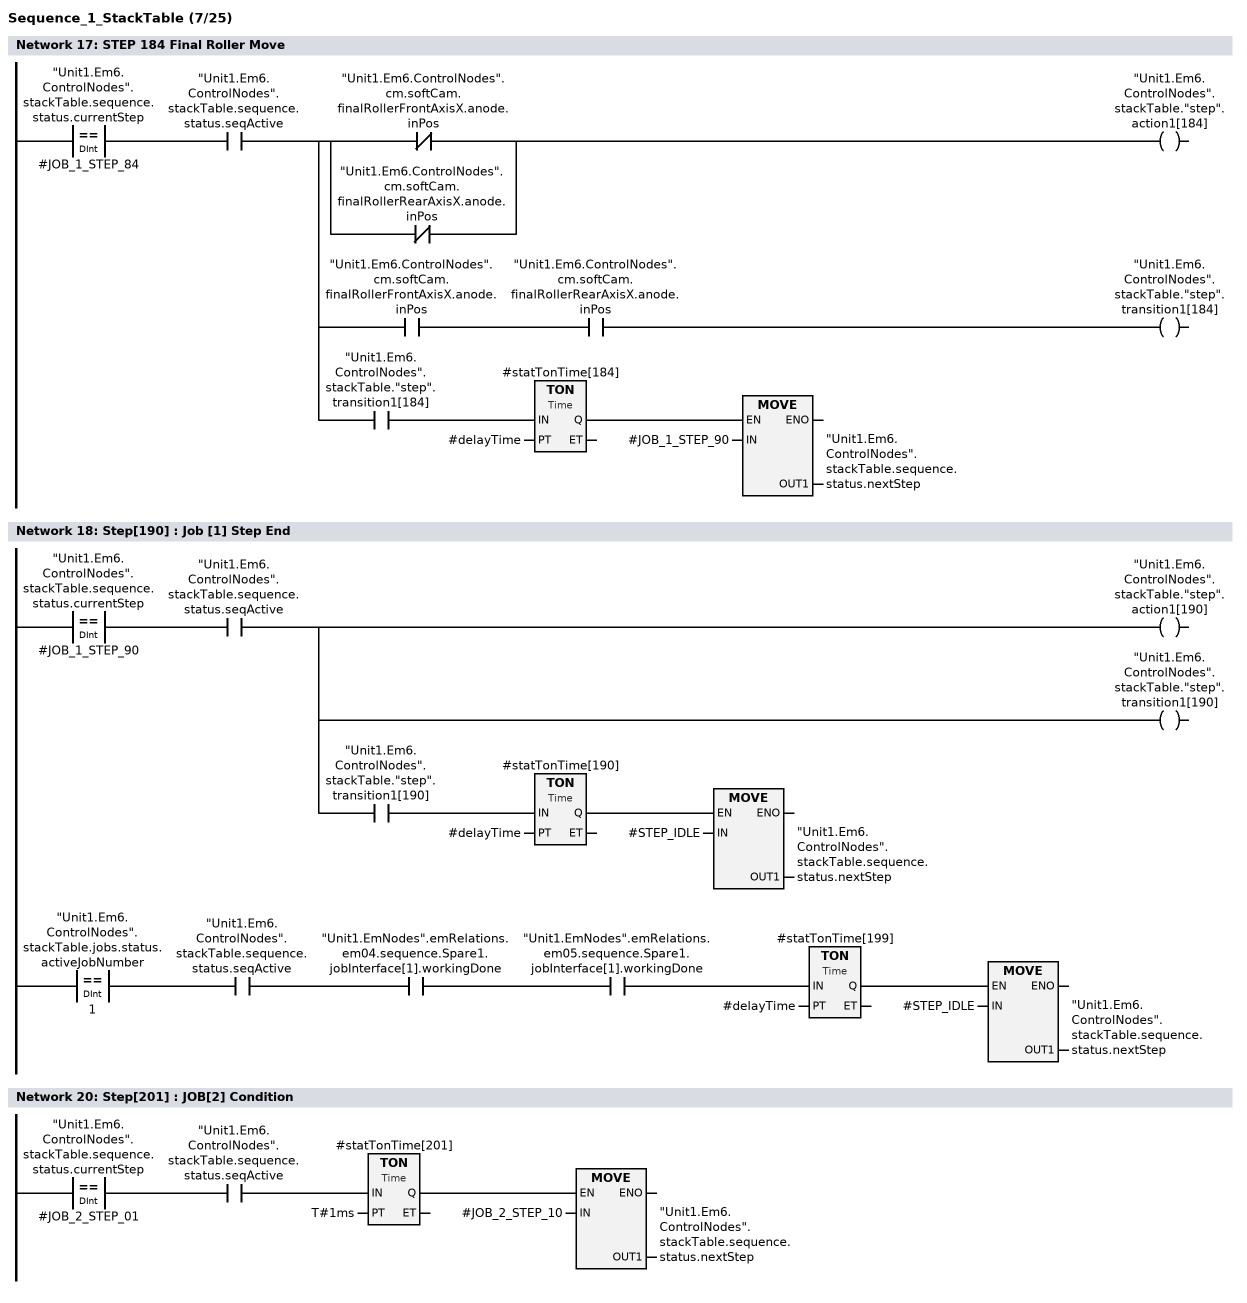
   RUNG wire#powerrail
      { S7_Templates := "SrcType := DInt" } EQ_Contact(in1 := "Unit1.Em6.ControlNodes".stackTable.sequence.status.currentStep, in2 := #JOB_1_STEP_84)
      Contact( "Unit1.Em6.ControlNodes".stackTable.sequence.status.seqActive )
      wire#w1
      I_Contact( "Unit1.Em6.ControlNodes".cm.softCam.finalRollerFrontAxisX.anode.inPos )
      wire#w2
      Coil( "Unit1.Em6.ControlNodes".stackTable."step".action1[184] )
   END_RUNG
   RUNG wire#w1
      I_Contact( "Unit1.Em6.ControlNodes".cm.softCam.finalRollerRearAxisX.anode.inPos )
   END_RUNG wire#w2
   RUNG wire#w1
      Contact( "Unit1.Em6.ControlNodes".cm.softCam.finalRollerFrontAxisX.anode.inPos )
      Contact( "Unit1.Em6.ControlNodes".cm.softCam.finalRollerRearAxisX.anode.inPos )
      Coil( "Unit1.Em6.ControlNodes".stackTable."step".transition1[184] )
   END_RUNG
   RUNG wire#w1
      Contact( "Unit1.Em6.ControlNodes".stackTable."step".transition1[184] )
      { S7_Templates := "time_type := Time" } #statTonTime[184].TON(pt := #delayTime, et =>)
      Move(in := #JOB_1_STEP_90, out1 => "Unit1.Em6.ControlNodes".stackTable.sequence.status.nextStep)
   END_RUNG
   // the same network as SCL:
   #_w1 := ("Unit1.Em6.ControlNodes".stackTable.sequence.status.currentStep = #JOB_1_STEP_84) AND "Unit1.Em6.ControlNodes".stackTable.sequence.status.seqActive;
   "Unit1.Em6.ControlNodes".stackTable."step".action1[184] := #_w1 AND (NOT "Unit1.Em6.ControlNodes".cm.softCam.finalRollerFrontAxisX.anode.inPos OR NOT "Unit1.Em6.ControlNodes".cm.softCam.finalRollerRearAxisX.anode.inPos);
   "Unit1.Em6.ControlNodes".stackTable."step".transition1[184] := #_w1 AND "Unit1.Em6.ControlNodes".cm.softCam.finalRollerFrontAxisX.anode.inPos AND "Unit1.Em6.ControlNodes".cm.softCam.finalRollerRearAxisX.anode.inPos;
   #statTonTime[184].TON(IN := #_w1 AND "Unit1.Em6.ControlNodes".stackTable."step".transition1[184],
                         PT := #delayTime);
   IF #statTonTime[184].Q THEN
       "Unit1.Em6.ControlNodes".stackTable.sequence.status.nextStep := #JOB_1_STEP_90;
   END_IF;
END_REGION

REGION Network 18: Step[190] : Job [1] Step End
   RUNG wire#powerrail
      { S7_Templates := "SrcType := DInt" } EQ_Contact(in1 := "Unit1.Em6.ControlNodes".stackTable.sequence.status.currentStep, in2 := #JOB_1_STEP_90)
      Contact( "Unit1.Em6.ControlNodes".stackTable.sequence.status.seqActive )
      wire#w1
      Coil( "Unit1.Em6.ControlNodes".stackTable."step".action1[190] )
   END_RUNG
   RUNG wire#w1
      Coil( "Unit1.Em6.ControlNodes".stackTable."step".transition1[190] )
   END_RUNG
   RUNG wire#w1
      Contact( "Unit1.Em6.ControlNodes".stackTable."step".transition1[190] )
      { S7_Templates := "time_type := Time" } #statTonTime[190].TON(pt := #delayTime, et =>)
      Move(in := #STEP_IDLE, out1 => "Unit1.Em6.ControlNodes".stackTable.sequence.status.nextStep)
   END_RUNG
   RUNG wire#powerrail
      { S7_Templates := "SrcType := DInt" } EQ_Contact(in1 := "Unit1.Em6.ControlNodes".stackTable.jobs.status.activeJobNumber, in2 := 1)
      Contact( "Unit1.Em6.ControlNodes".stackTable.sequence.status.seqActive )
      Contact( "Unit1.EmNodes".emRelations.em04.sequence.Spare1.jobInterface[1].workingDone )
      Contact( "Unit1.EmNodes".emRelations.em05.sequence.Spare1.jobInterface[1].workingDone )
      { S7_Templates := "time_type := Time" } #statTonTime[199].TON(pt := #delayTime, et =>)
      Move(in := #STEP_IDLE, out1 => "Unit1.Em6.ControlNodes".stackTable.sequence.status.nextStep)
   END_RUNG
   // the same network as SCL:
   "Unit1.Em6.ControlNodes".stackTable."step".action1[190] := ("Unit1.Em6.ControlNodes".stackTable.sequence.status.currentStep = #JOB_1_STEP_90) AND "Unit1.Em6.ControlNodes".stackTable.sequence.status.seqActive;
   "Unit1.Em6.ControlNodes".stackTable."step".transition1[190] := ("Unit1.Em6.ControlNodes".stackTable.sequence.status.currentStep = #JOB_1_STEP_90) AND "Unit1.Em6.ControlNodes".stackTable.sequence.status.seqActive;
   #statTonTime[190].TON(IN := ("Unit1.Em6.ControlNodes".stackTable.sequence.status.currentStep = #JOB_1_STEP_90) AND "Unit1.Em6.ControlNodes".stackTable.sequence.status.seqActive AND "Unit1.Em6.ControlNodes".stackTable."step".transition1[190],
                         PT := #delayTime);
   IF #statTonTime[190].Q THEN
       "Unit1.Em6.ControlNodes".stackTable.sequence.status.nextStep := #STEP_IDLE;
   END_IF;
   #statTonTime[199].TON(IN := ("Unit1.Em6.ControlNodes".stackTable.jobs.status.activeJobNumber = 1) AND "Unit1.Em6.ControlNodes".stackTable.sequence.status.seqActive AND "Unit1.EmNodes".emRelations.em04.sequence.Spare1.jobInterface[1].workingDone AND "Unit1.EmNodes".emRelations.em05.sequence.Spare1.jobInterface[1].workingDone,
                         PT := #delayTime);
   IF #statTonTime[199].Q THEN
       "Unit1.Em6.ControlNodes".stackTable.sequence.status.nextStep := #STEP_IDLE;
   END_IF;
END_REGION

REGION Network 19: ******************** JOB[2] Motion Auto ********************
END_REGION

REGION Network 20: Step[201] : JOB[2] Condition
   RUNG wire#powerrail
      { S7_Templates := "SrcType := DInt" } EQ_Contact(in1 := "Unit1.Em6.ControlNodes".stackTable.sequence.status.currentStep, in2 := #JOB_2_STEP_01)
      Contact( "Unit1.Em6.ControlNodes".stackTable.sequence.status.seqActive )
      { S7_Templates := "time_type := Time" } #statTonTime[201].TON(pt := T#1ms, et =>)
      Move(in := #JOB_2_STEP_10, out1 => "Unit1.Em6.ControlNodes".stackTable.sequence.status.nextStep)
   END_RUNG
   // the same network as SCL:
   #statTonTime[201].TON(IN := ("Unit1.Em6.ControlNodes".stackTable.sequence.status.currentStep = #JOB_2_STEP_01) AND "Unit1.Em6.ControlNodes".stackTable.sequence.status.seqActive,
                         PT := T#1ms);
   IF #statTonTime[201].Q THEN
       "Unit1.Em6.ControlNodes".stackTable.sequence.status.nextStep := #JOB_2_STEP_10;
   END_IF;
END_REGION

REGION Network 21: Step[210] : Vision Start
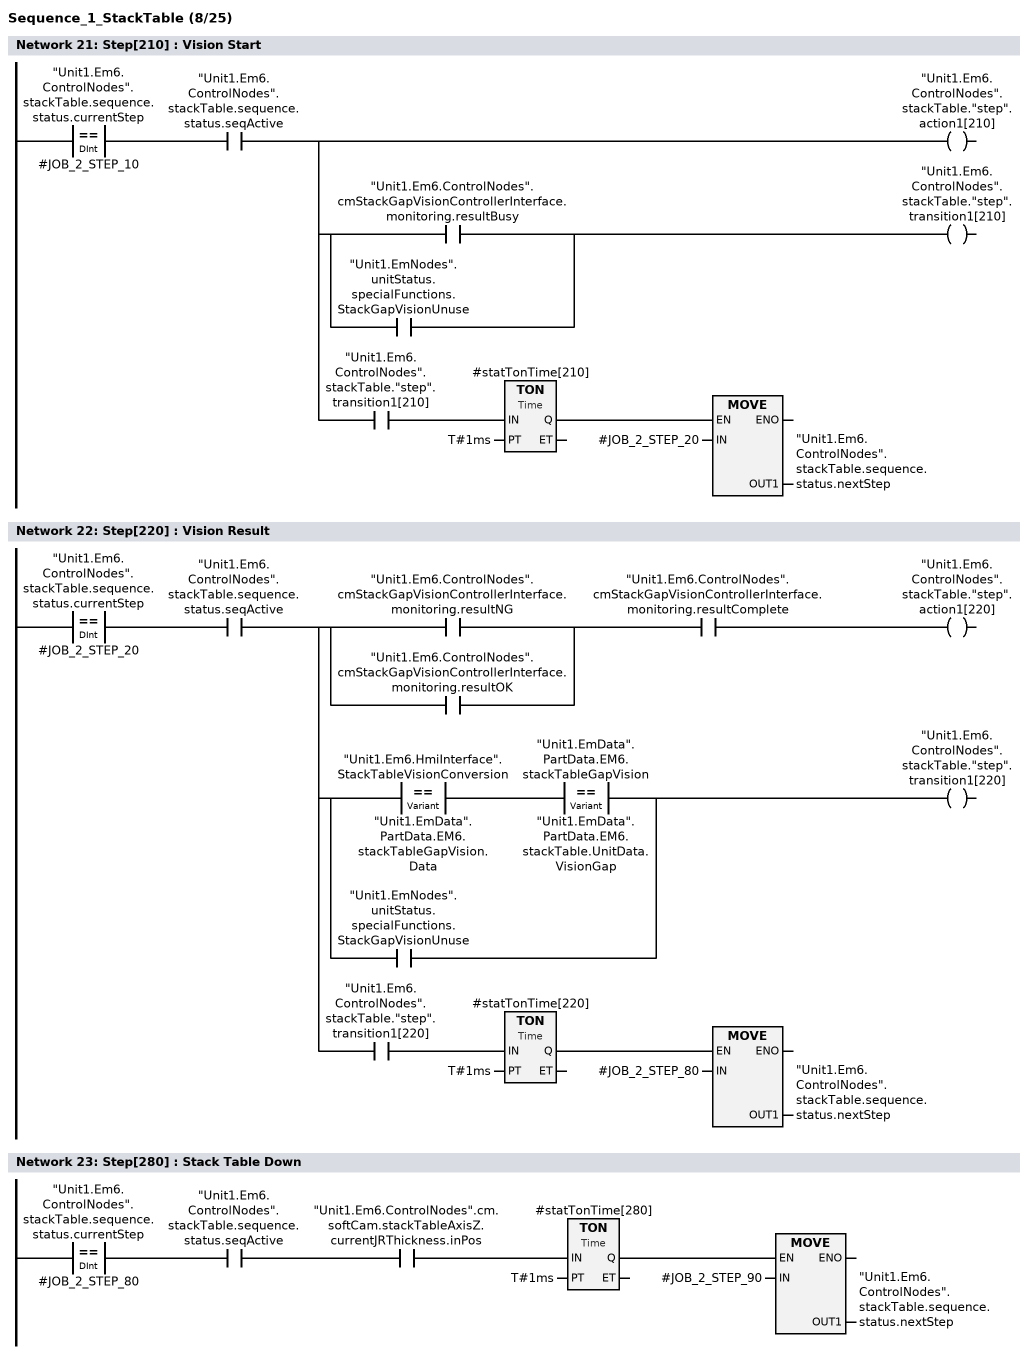
   RUNG wire#powerrail
      { S7_Templates := "SrcType := DInt" } EQ_Contact(in1 := "Unit1.Em6.ControlNodes".stackTable.sequence.status.currentStep, in2 := #JOB_2_STEP_10)
      Contact( "Unit1.Em6.ControlNodes".stackTable.sequence.status.seqActive )
      wire#w1
      Coil( "Unit1.Em6.ControlNodes".stackTable."step".action1[210] )
   END_RUNG
   RUNG wire#w1
      Contact( "Unit1.Em6.ControlNodes".cmStackGapVisionControllerInterface.monitoring.resultBusy )
      wire#w2
      Coil( "Unit1.Em6.ControlNodes".stackTable."step".transition1[210] )
   END_RUNG
   RUNG wire#w1
      Contact( "Unit1.EmNodes".unitStatus.specialFunctions.StackGapVisionUnuse )
   END_RUNG wire#w2
   RUNG wire#w1
      Contact( "Unit1.Em6.ControlNodes".stackTable."step".transition1[210] )
      { S7_Templates := "time_type := Time" } #statTonTime[210].TON(pt := T#1ms, et =>)
      Move(in := #JOB_2_STEP_20, out1 => "Unit1.Em6.ControlNodes".stackTable.sequence.status.nextStep)
   END_RUNG
   // the same network as SCL:
   "Unit1.Em6.ControlNodes".stackTable."step".action1[210] := ("Unit1.Em6.ControlNodes".stackTable.sequence.status.currentStep = #JOB_2_STEP_10) AND "Unit1.Em6.ControlNodes".stackTable.sequence.status.seqActive;
   "Unit1.Em6.ControlNodes".stackTable."step".transition1[210] := ("Unit1.Em6.ControlNodes".stackTable.sequence.status.currentStep = #JOB_2_STEP_10) AND "Unit1.Em6.ControlNodes".stackTable.sequence.status.seqActive AND ("Unit1.Em6.ControlNodes".cmStackGapVisionControllerInterface.monitoring.resultBusy OR "Unit1.EmNodes".unitStatus.specialFunctions.StackGapVisionUnuse);
   #statTonTime[210].TON(IN := ("Unit1.Em6.ControlNodes".stackTable.sequence.status.currentStep = #JOB_2_STEP_10) AND "Unit1.Em6.ControlNodes".stackTable.sequence.status.seqActive AND "Unit1.Em6.ControlNodes".stackTable."step".transition1[210],
                         PT := T#1ms);
   IF #statTonTime[210].Q THEN
       "Unit1.Em6.ControlNodes".stackTable.sequence.status.nextStep := #JOB_2_STEP_20;
   END_IF;
END_REGION

REGION Network 22: Step[220] : Vision Result
   RUNG wire#powerrail
      { S7_Templates := "SrcType := DInt" } EQ_Contact(in1 := "Unit1.Em6.ControlNodes".stackTable.sequence.status.currentStep, in2 := #JOB_2_STEP_20)
      Contact( "Unit1.Em6.ControlNodes".stackTable.sequence.status.seqActive )
      wire#w1
      Contact( "Unit1.Em6.ControlNodes".cmStackGapVisionControllerInterface.monitoring.resultNG )
      wire#w2
      Contact( "Unit1.Em6.ControlNodes".cmStackGapVisionControllerInterface.monitoring.resultComplete )
      Coil( "Unit1.Em6.ControlNodes".stackTable."step".action1[220] )
   END_RUNG
   RUNG wire#w1
      Contact( "Unit1.Em6.ControlNodes".cmStackGapVisionControllerInterface.monitoring.resultOK )
   END_RUNG wire#w2
   RUNG wire#w1
      { S7_Templates := "SrcType := Variant" } EQ_Contact(in1 := "Unit1.Em6.HmiInterface".StackTableVisionConversion, in2 := "Unit1.EmData".PartData.EM6.stackTableGapVision.Data)
      { S7_Templates := "SrcType := Variant" } EQ_Contact(in1 := "Unit1.EmData".PartData.EM6.stackTableGapVision, in2 := "Unit1.EmData".PartData.EM6.stackTable.UnitData.VisionGap)
      wire#w3
      Coil( "Unit1.Em6.ControlNodes".stackTable."step".transition1[220] )
   END_RUNG
   RUNG wire#w1
      Contact( "Unit1.EmNodes".unitStatus.specialFunctions.StackGapVisionUnuse )
   END_RUNG wire#w3
   RUNG wire#w1
      Contact( "Unit1.Em6.ControlNodes".stackTable."step".transition1[220] )
      { S7_Templates := "time_type := Time" } #statTonTime[220].TON(pt := T#1ms, et =>)
      Move(in := #JOB_2_STEP_80, out1 => "Unit1.Em6.ControlNodes".stackTable.sequence.status.nextStep)
   END_RUNG
   // the same network as SCL:
   #_w1 := ("Unit1.Em6.ControlNodes".stackTable.sequence.status.currentStep = #JOB_2_STEP_20) AND "Unit1.Em6.ControlNodes".stackTable.sequence.status.seqActive;
   "Unit1.Em6.ControlNodes".stackTable."step".action1[220] := #_w1 AND ("Unit1.Em6.ControlNodes".cmStackGapVisionControllerInterface.monitoring.resultNG OR "Unit1.Em6.ControlNodes".cmStackGapVisionControllerInterface.monitoring.resultOK) AND "Unit1.Em6.ControlNodes".cmStackGapVisionControllerInterface.monitoring.resultComplete;
   "Unit1.Em6.ControlNodes".stackTable."step".transition1[220] := #_w1 AND ((("Unit1.Em6.HmiInterface".StackTableVisionConversion = "Unit1.EmData".PartData.EM6.stackTableGapVision.Data) AND ("Unit1.EmData".PartData.EM6.stackTableGapVision = "Unit1.EmData".PartData.EM6.stackTable.UnitData.VisionGap)) OR "Unit1.EmNodes".unitStatus.specialFunctions.StackGapVisionUnuse);
   #statTonTime[220].TON(IN := #_w1 AND "Unit1.Em6.ControlNodes".stackTable."step".transition1[220],
                         PT := T#1ms);
   IF #statTonTime[220].Q THEN
       "Unit1.Em6.ControlNodes".stackTable.sequence.status.nextStep := #JOB_2_STEP_80;
   END_IF;
END_REGION

REGION Network 23: Step[280] : Stack Table Down
   RUNG wire#powerrail
      { S7_Templates := "SrcType := DInt" } EQ_Contact(in1 := "Unit1.Em6.ControlNodes".stackTable.sequence.status.currentStep, in2 := #JOB_2_STEP_80)
      Contact( "Unit1.Em6.ControlNodes".stackTable.sequence.status.seqActive )
      Contact( "Unit1.Em6.ControlNodes".cm.softCam.stackTableAxisZ.currentJRThickness.inPos )
      { S7_Templates := "time_type := Time" } #statTonTime[280].TON(pt := T#1ms, et =>)
      Move(in := #JOB_2_STEP_90, out1 => "Unit1.Em6.ControlNodes".stackTable.sequence.status.nextStep)
   END_RUNG
   // the same network as SCL:
   #statTonTime[280].TON(IN := ("Unit1.Em6.ControlNodes".stackTable.sequence.status.currentStep = #JOB_2_STEP_80) AND "Unit1.Em6.ControlNodes".stackTable.sequence.status.seqActive AND "Unit1.Em6.ControlNodes".cm.softCam.stackTableAxisZ.currentJRThickness.inPos,
                         PT := T#1ms);
   IF #statTonTime[280].Q THEN
       "Unit1.Em6.ControlNodes".stackTable.sequence.status.nextStep := #JOB_2_STEP_90;
   END_IF;
END_REGION

REGION Network 24: Step[290] : JOB[2] Step End
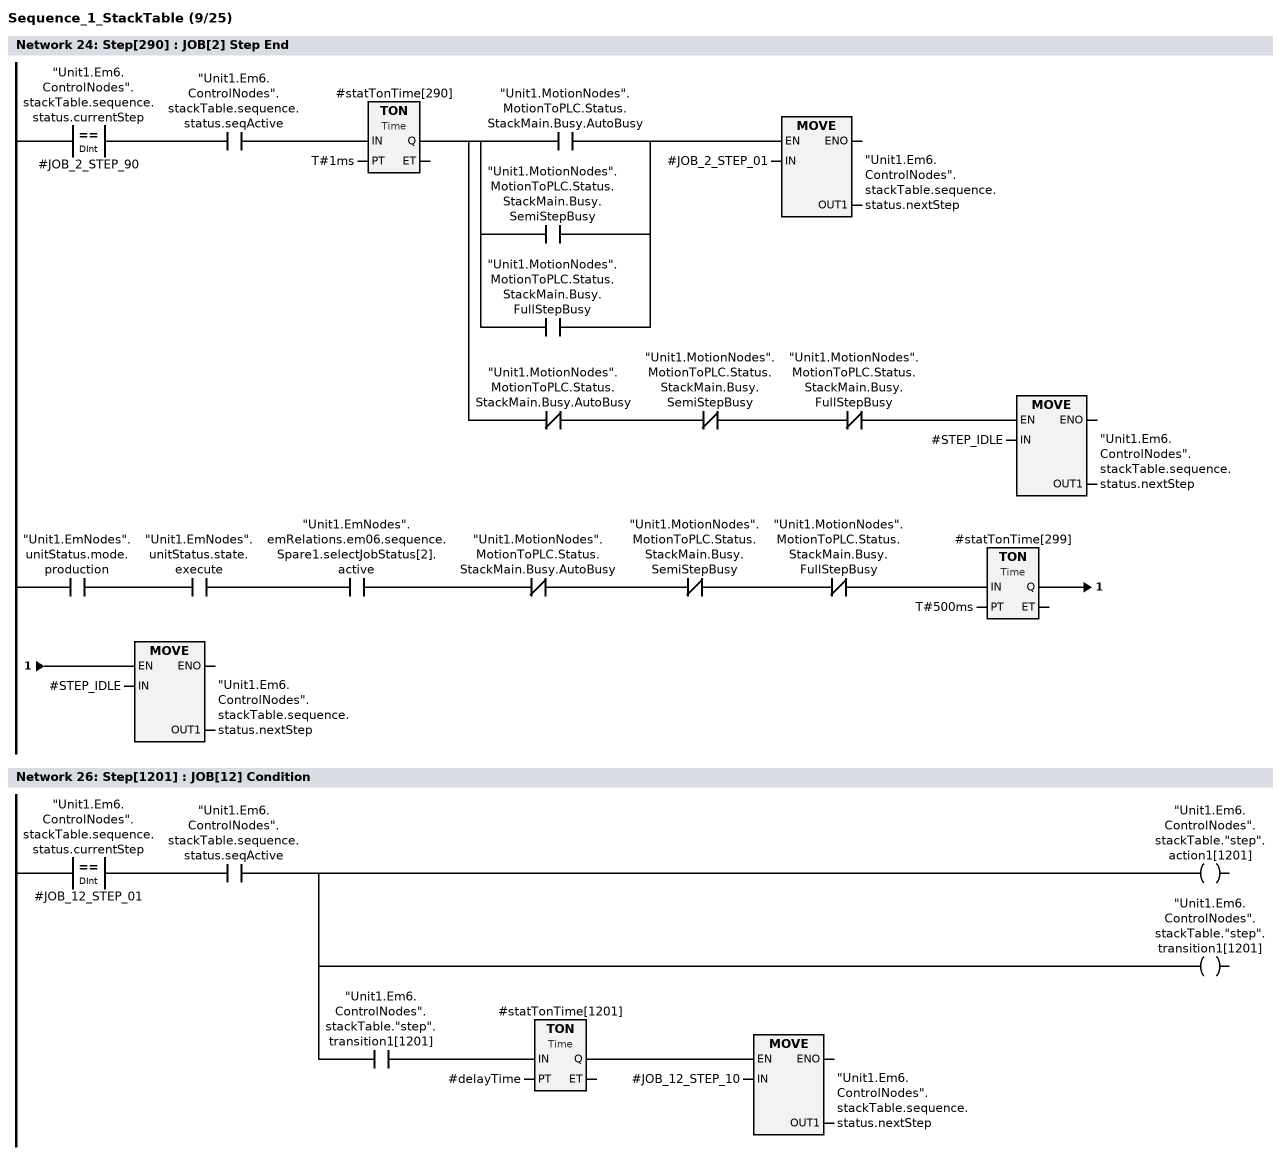
   RUNG wire#powerrail
      { S7_Templates := "SrcType := DInt" } EQ_Contact(in1 := "Unit1.Em6.ControlNodes".stackTable.sequence.status.currentStep, in2 := #JOB_2_STEP_90)
      Contact( "Unit1.Em6.ControlNodes".stackTable.sequence.status.seqActive )
      { S7_Templates := "time_type := Time" } #statTonTime[290].TON(pt := T#1ms, et =>)
      wire#w1
      Contact( "Unit1.MotionNodes".MotionToPLC.Status.StackMain.Busy.AutoBusy )
      wire#w2
      Move(in := #JOB_2_STEP_01, out1 => "Unit1.Em6.ControlNodes".stackTable.sequence.status.nextStep)
   END_RUNG
   RUNG wire#w1
      Contact( "Unit1.MotionNodes".MotionToPLC.Status.StackMain.Busy.SemiStepBusy )
   END_RUNG wire#w2
   RUNG wire#w1
      Contact( "Unit1.MotionNodes".MotionToPLC.Status.StackMain.Busy.FullStepBusy )
   END_RUNG wire#w2
   RUNG wire#w1
      I_Contact( "Unit1.MotionNodes".MotionToPLC.Status.StackMain.Busy.AutoBusy )
      I_Contact( "Unit1.MotionNodes".MotionToPLC.Status.StackMain.Busy.SemiStepBusy )
      I_Contact( "Unit1.MotionNodes".MotionToPLC.Status.StackMain.Busy.FullStepBusy )
      Move(in := #STEP_IDLE, out1 => "Unit1.Em6.ControlNodes".stackTable.sequence.status.nextStep)
   END_RUNG
   RUNG wire#powerrail
      Contact( "Unit1.EmNodes".unitStatus.mode.production )
      Contact( "Unit1.EmNodes".unitStatus.state.execute )
      Contact( "Unit1.EmNodes".emRelations.em06.sequence.Spare1.selectJobStatus[2].active )
      I_Contact( "Unit1.MotionNodes".MotionToPLC.Status.StackMain.Busy.AutoBusy )
      I_Contact( "Unit1.MotionNodes".MotionToPLC.Status.StackMain.Busy.SemiStepBusy )
      I_Contact( "Unit1.MotionNodes".MotionToPLC.Status.StackMain.Busy.FullStepBusy )
      { S7_Templates := "time_type := Time" } #statTonTime[299].TON(pt := T#500ms, et =>)
      Move(in := #STEP_IDLE, out1 => "Unit1.Em6.ControlNodes".stackTable.sequence.status.nextStep)
   END_RUNG
   // the same network as SCL:
   #statTonTime[290].TON(IN := ("Unit1.Em6.ControlNodes".stackTable.sequence.status.currentStep = #JOB_2_STEP_90) AND "Unit1.Em6.ControlNodes".stackTable.sequence.status.seqActive,
                         PT := T#1ms);
   IF #statTonTime[290].Q AND ("Unit1.MotionNodes".MotionToPLC.Status.StackMain.Busy.AutoBusy OR "Unit1.MotionNodes".MotionToPLC.Status.StackMain.Busy.SemiStepBusy OR "Unit1.MotionNodes".MotionToPLC.Status.StackMain.Busy.FullStepBusy) THEN
       "Unit1.Em6.ControlNodes".stackTable.sequence.status.nextStep := #JOB_2_STEP_01;
   END_IF;
   IF #statTonTime[290].Q AND NOT "Unit1.MotionNodes".MotionToPLC.Status.StackMain.Busy.AutoBusy AND NOT "Unit1.MotionNodes".MotionToPLC.Status.StackMain.Busy.SemiStepBusy AND NOT "Unit1.MotionNodes".MotionToPLC.Status.StackMain.Busy.FullStepBusy THEN
       "Unit1.Em6.ControlNodes".stackTable.sequence.status.nextStep := #STEP_IDLE;
   END_IF;
   #statTonTime[299].TON(IN := "Unit1.EmNodes".unitStatus.mode.production AND "Unit1.EmNodes".unitStatus.state.execute AND "Unit1.EmNodes".emRelations.em06.sequence.Spare1.selectJobStatus[2].active AND NOT "Unit1.MotionNodes".MotionToPLC.Status.StackMain.Busy.AutoBusy AND NOT "Unit1.MotionNodes".MotionToPLC.Status.StackMain.Busy.SemiStepBusy AND NOT "Unit1.MotionNodes".MotionToPLC.Status.StackMain.Busy.FullStepBusy,
                         PT := T#500ms);
   IF #statTonTime[299].Q THEN
       "Unit1.Em6.ControlNodes".stackTable.sequence.status.nextStep := #STEP_IDLE;
   END_IF;
END_REGION

REGION Network 25: ******************** JOB[12] Final Roller Move [Cathode → Anode] ********************
END_REGION

REGION Network 26: Step[1201] : JOB[12] Condition
   RUNG wire#powerrail
      { S7_Templates := "SrcType := DInt" } EQ_Contact(in1 := "Unit1.Em6.ControlNodes".stackTable.sequence.status.currentStep, in2 := #JOB_12_STEP_01)
      Contact( "Unit1.Em6.ControlNodes".stackTable.sequence.status.seqActive )
      wire#w1
      Coil( "Unit1.Em6.ControlNodes".stackTable."step".action1[1201] )
   END_RUNG
   RUNG wire#w1
      Coil( "Unit1.Em6.ControlNodes".stackTable."step".transition1[1201] )
   END_RUNG
   RUNG wire#w1
      Contact( "Unit1.Em6.ControlNodes".stackTable."step".transition1[1201] )
      { S7_Templates := "time_type := Time" } #statTonTime[1201].TON(pt := #delayTime, et =>)
      Move(in := #JOB_12_STEP_10, out1 => "Unit1.Em6.ControlNodes".stackTable.sequence.status.nextStep)
   END_RUNG
   // the same network as SCL:
   "Unit1.Em6.ControlNodes".stackTable."step".action1[1201] := ("Unit1.Em6.ControlNodes".stackTable.sequence.status.currentStep = #JOB_12_STEP_01) AND "Unit1.Em6.ControlNodes".stackTable.sequence.status.seqActive;
   "Unit1.Em6.ControlNodes".stackTable."step".transition1[1201] := ("Unit1.Em6.ControlNodes".stackTable.sequence.status.currentStep = #JOB_12_STEP_01) AND "Unit1.Em6.ControlNodes".stackTable.sequence.status.seqActive;
   #statTonTime[1201].TON(IN := ("Unit1.Em6.ControlNodes".stackTable.sequence.status.currentStep = #JOB_12_STEP_01) AND "Unit1.Em6.ControlNodes".stackTable.sequence.status.seqActive AND "Unit1.Em6.ControlNodes".stackTable."step".transition1[1201],
                          PT := #delayTime);
   IF #statTonTime[1201].Q THEN
       "Unit1.Em6.ControlNodes".stackTable.sequence.status.nextStep := #JOB_12_STEP_10;
   END_IF;
END_REGION

REGION Network 27: Step[1210] : FinalRoller X-Axis Anode Pos
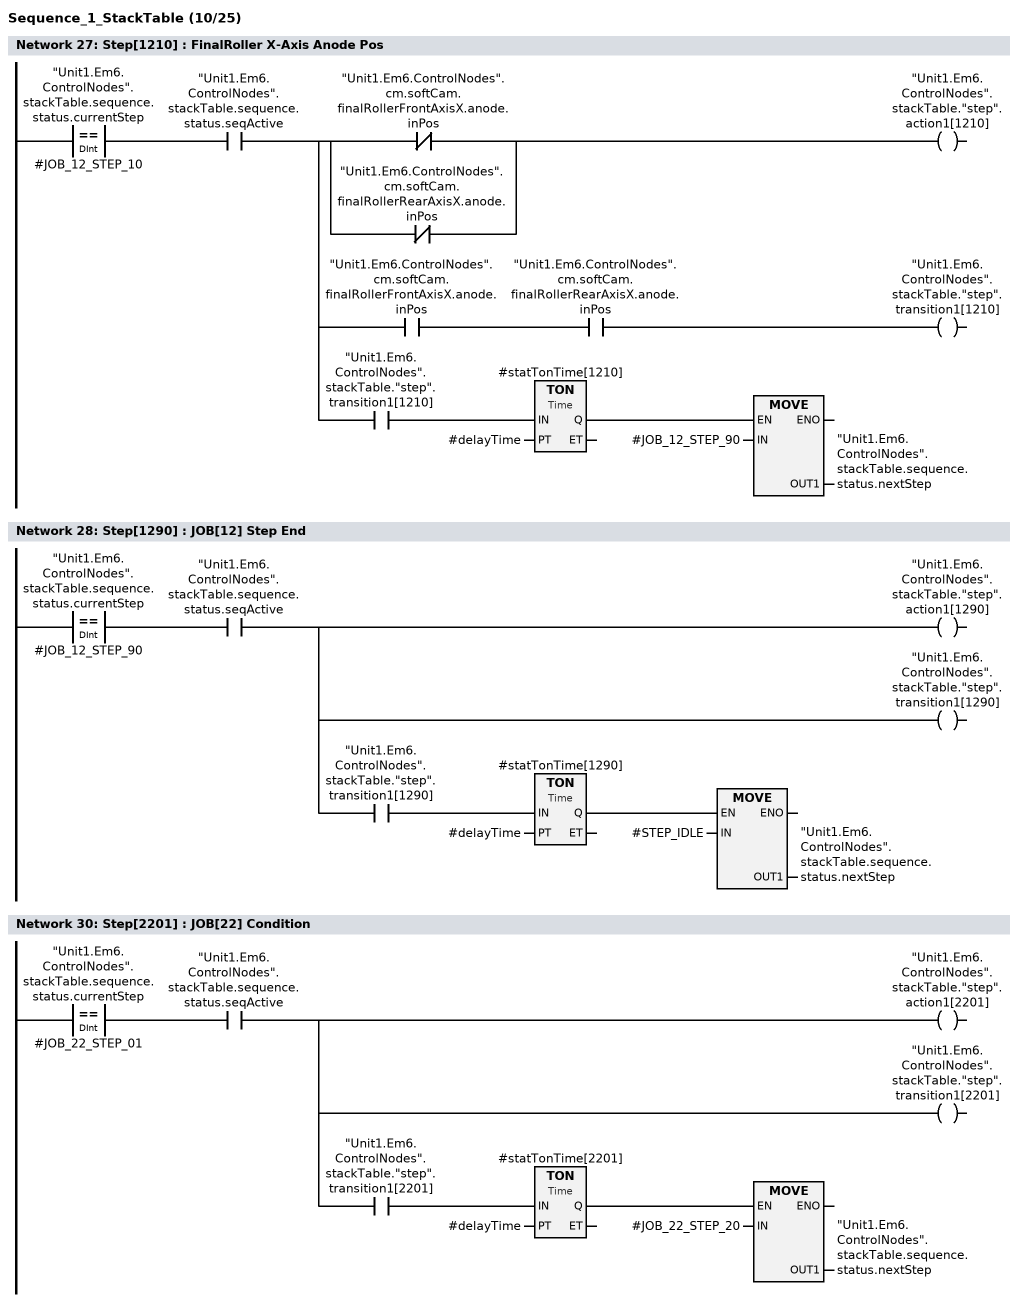
   RUNG wire#powerrail
      { S7_Templates := "SrcType := DInt" } EQ_Contact(in1 := "Unit1.Em6.ControlNodes".stackTable.sequence.status.currentStep, in2 := #JOB_12_STEP_10)
      Contact( "Unit1.Em6.ControlNodes".stackTable.sequence.status.seqActive )
      wire#w1
      I_Contact( "Unit1.Em6.ControlNodes".cm.softCam.finalRollerFrontAxisX.anode.inPos )
      wire#w2
      Coil( "Unit1.Em6.ControlNodes".stackTable."step".action1[1210] )
   END_RUNG
   RUNG wire#w1
      I_Contact( "Unit1.Em6.ControlNodes".cm.softCam.finalRollerRearAxisX.anode.inPos )
   END_RUNG wire#w2
   RUNG wire#w1
      Contact( "Unit1.Em6.ControlNodes".cm.softCam.finalRollerFrontAxisX.anode.inPos )
      Contact( "Unit1.Em6.ControlNodes".cm.softCam.finalRollerRearAxisX.anode.inPos )
      Coil( "Unit1.Em6.ControlNodes".stackTable."step".transition1[1210] )
   END_RUNG
   RUNG wire#w1
      Contact( "Unit1.Em6.ControlNodes".stackTable."step".transition1[1210] )
      { S7_Templates := "time_type := Time" } #statTonTime[1210].TON(pt := #delayTime, et =>)
      Move(in := #JOB_12_STEP_90, out1 => "Unit1.Em6.ControlNodes".stackTable.sequence.status.nextStep)
   END_RUNG
   // the same network as SCL:
   #_w1 := ("Unit1.Em6.ControlNodes".stackTable.sequence.status.currentStep = #JOB_12_STEP_10) AND "Unit1.Em6.ControlNodes".stackTable.sequence.status.seqActive;
   "Unit1.Em6.ControlNodes".stackTable."step".action1[1210] := #_w1 AND (NOT "Unit1.Em6.ControlNodes".cm.softCam.finalRollerFrontAxisX.anode.inPos OR NOT "Unit1.Em6.ControlNodes".cm.softCam.finalRollerRearAxisX.anode.inPos);
   "Unit1.Em6.ControlNodes".stackTable."step".transition1[1210] := #_w1 AND "Unit1.Em6.ControlNodes".cm.softCam.finalRollerFrontAxisX.anode.inPos AND "Unit1.Em6.ControlNodes".cm.softCam.finalRollerRearAxisX.anode.inPos;
   #statTonTime[1210].TON(IN := #_w1 AND "Unit1.Em6.ControlNodes".stackTable."step".transition1[1210],
                          PT := #delayTime);
   IF #statTonTime[1210].Q THEN
       "Unit1.Em6.ControlNodes".stackTable.sequence.status.nextStep := #JOB_12_STEP_90;
   END_IF;
END_REGION

REGION Network 28: Step[1290] : JOB[12] Step End
   RUNG wire#powerrail
      { S7_Templates := "SrcType := DInt" } EQ_Contact(in1 := "Unit1.Em6.ControlNodes".stackTable.sequence.status.currentStep, in2 := #JOB_12_STEP_90)
      Contact( "Unit1.Em6.ControlNodes".stackTable.sequence.status.seqActive )
      wire#w1
      Coil( "Unit1.Em6.ControlNodes".stackTable."step".action1[1290] )
   END_RUNG
   RUNG wire#w1
      Coil( "Unit1.Em6.ControlNodes".stackTable."step".transition1[1290] )
   END_RUNG
   RUNG wire#w1
      Contact( "Unit1.Em6.ControlNodes".stackTable."step".transition1[1290] )
      { S7_Templates := "time_type := Time" } #statTonTime[1290].TON(pt := #delayTime, et =>)
      Move(in := #STEP_IDLE, out1 => "Unit1.Em6.ControlNodes".stackTable.sequence.status.nextStep)
   END_RUNG
   // the same network as SCL:
   "Unit1.Em6.ControlNodes".stackTable."step".action1[1290] := ("Unit1.Em6.ControlNodes".stackTable.sequence.status.currentStep = #JOB_12_STEP_90) AND "Unit1.Em6.ControlNodes".stackTable.sequence.status.seqActive;
   "Unit1.Em6.ControlNodes".stackTable."step".transition1[1290] := ("Unit1.Em6.ControlNodes".stackTable.sequence.status.currentStep = #JOB_12_STEP_90) AND "Unit1.Em6.ControlNodes".stackTable.sequence.status.seqActive;
   #statTonTime[1290].TON(IN := ("Unit1.Em6.ControlNodes".stackTable.sequence.status.currentStep = #JOB_12_STEP_90) AND "Unit1.Em6.ControlNodes".stackTable.sequence.status.seqActive AND "Unit1.Em6.ControlNodes".stackTable."step".transition1[1290],
                          PT := #delayTime);
   IF #statTonTime[1290].Q THEN
       "Unit1.Em6.ControlNodes".stackTable.sequence.status.nextStep := #STEP_IDLE;
   END_IF;
END_REGION

REGION Network 29: ******************** JOB[22] Anode Mendrel ********************
END_REGION

REGION Network 30: Step[2201] : JOB[22] Condition
   RUNG wire#powerrail
      { S7_Templates := "SrcType := DInt" } EQ_Contact(in1 := "Unit1.Em6.ControlNodes".stackTable.sequence.status.currentStep, in2 := #JOB_22_STEP_01)
      Contact( "Unit1.Em6.ControlNodes".stackTable.sequence.status.seqActive )
      wire#w1
      Coil( "Unit1.Em6.ControlNodes".stackTable."step".action1[2201] )
   END_RUNG
   RUNG wire#w1
      Coil( "Unit1.Em6.ControlNodes".stackTable."step".transition1[2201] )
   END_RUNG
   RUNG wire#w1
      Contact( "Unit1.Em6.ControlNodes".stackTable."step".transition1[2201] )
      { S7_Templates := "time_type := Time" } #statTonTime[2201].TON(pt := #delayTime, et =>)
      Move(in := #JOB_22_STEP_20, out1 => "Unit1.Em6.ControlNodes".stackTable.sequence.status.nextStep)
   END_RUNG
   // the same network as SCL:
   "Unit1.Em6.ControlNodes".stackTable."step".action1[2201] := ("Unit1.Em6.ControlNodes".stackTable.sequence.status.currentStep = #JOB_22_STEP_01) AND "Unit1.Em6.ControlNodes".stackTable.sequence.status.seqActive;
   "Unit1.Em6.ControlNodes".stackTable."step".transition1[2201] := ("Unit1.Em6.ControlNodes".stackTable.sequence.status.currentStep = #JOB_22_STEP_01) AND "Unit1.Em6.ControlNodes".stackTable.sequence.status.seqActive;
   #statTonTime[2201].TON(IN := ("Unit1.Em6.ControlNodes".stackTable.sequence.status.currentStep = #JOB_22_STEP_01) AND "Unit1.Em6.ControlNodes".stackTable.sequence.status.seqActive AND "Unit1.Em6.ControlNodes".stackTable."step".transition1[2201],
                          PT := #delayTime);
   IF #statTonTime[2201].Q THEN
       "Unit1.Em6.ControlNodes".stackTable.sequence.status.nextStep := #JOB_22_STEP_20;
   END_IF;
END_REGION

REGION Network 31: Step[2220] : A.Mendrel Y,Z-Axis Wait Pos
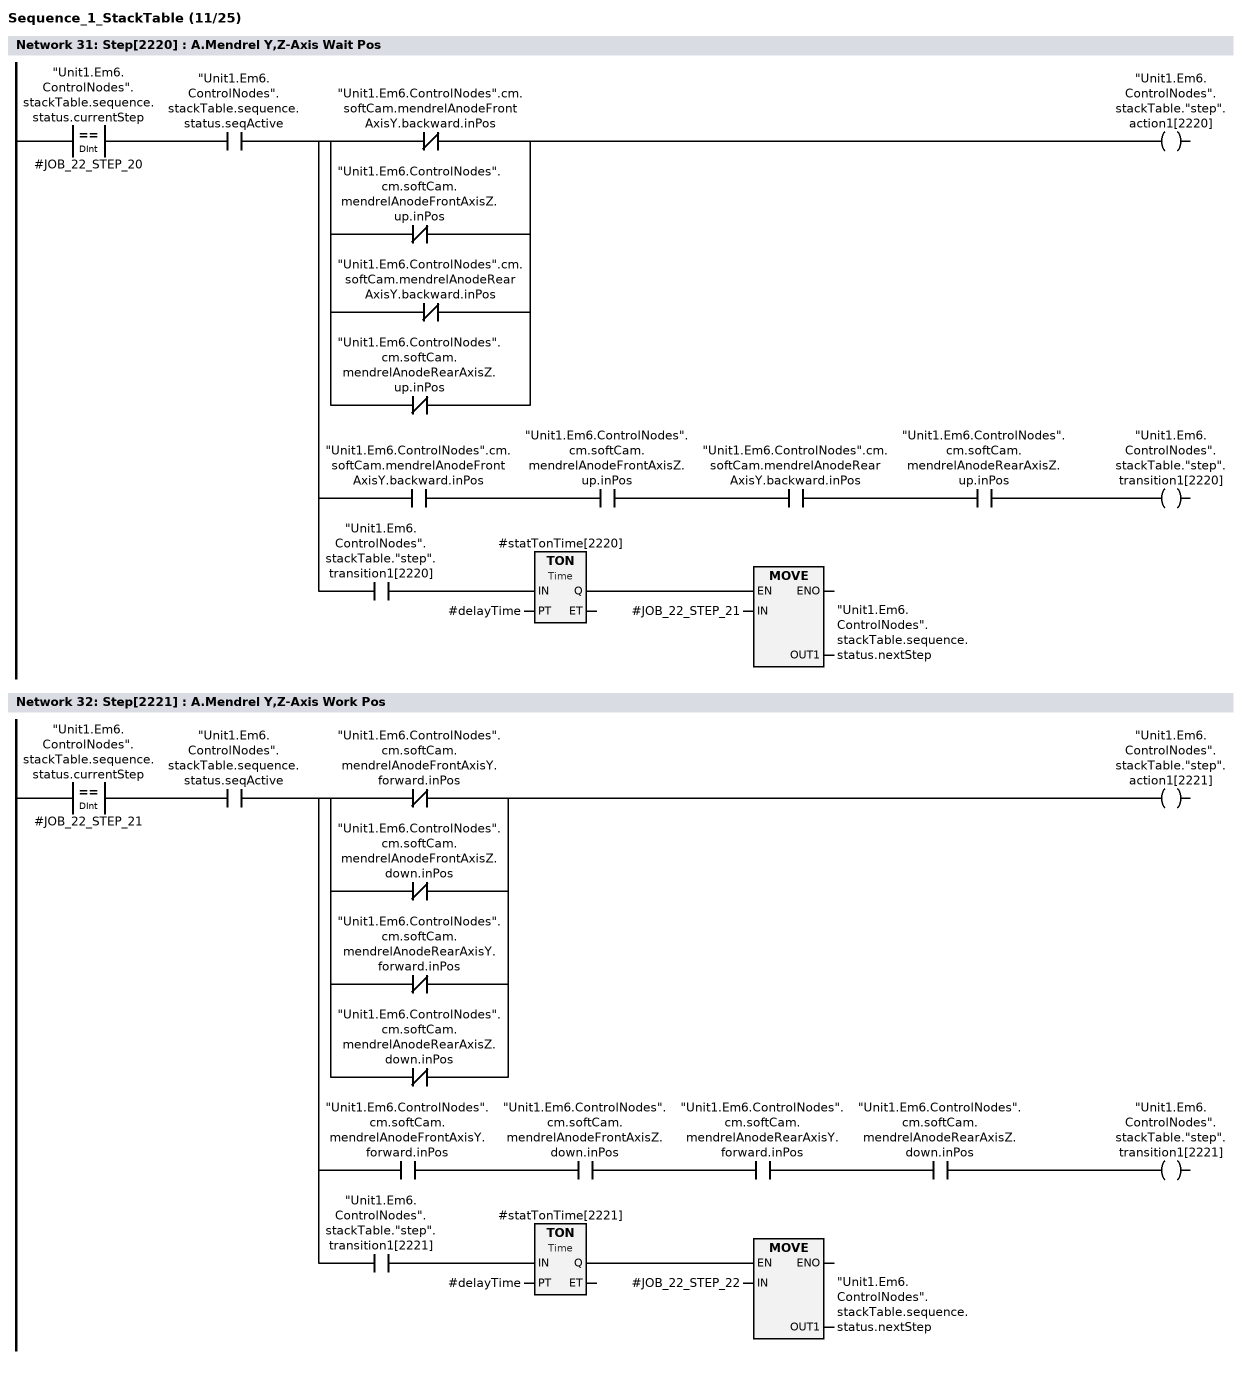
   RUNG wire#powerrail
      { S7_Templates := "SrcType := DInt" } EQ_Contact(in1 := "Unit1.Em6.ControlNodes".stackTable.sequence.status.currentStep, in2 := #JOB_22_STEP_20)
      Contact( "Unit1.Em6.ControlNodes".stackTable.sequence.status.seqActive )
      wire#w1
      I_Contact( "Unit1.Em6.ControlNodes".cm.softCam.mendrelAnodeFrontAxisY.backward.inPos )
      wire#w2
      Coil( "Unit1.Em6.ControlNodes".stackTable."step".action1[2220] )
   END_RUNG
   RUNG wire#w1
      I_Contact( "Unit1.Em6.ControlNodes".cm.softCam.mendrelAnodeFrontAxisZ.up.inPos )
   END_RUNG wire#w2
   RUNG wire#w1
      I_Contact( "Unit1.Em6.ControlNodes".cm.softCam.mendrelAnodeRearAxisY.backward.inPos )
   END_RUNG wire#w2
   RUNG wire#w1
      I_Contact( "Unit1.Em6.ControlNodes".cm.softCam.mendrelAnodeRearAxisZ.up.inPos )
   END_RUNG wire#w2
   RUNG wire#w1
      Contact( "Unit1.Em6.ControlNodes".cm.softCam.mendrelAnodeFrontAxisY.backward.inPos )
      Contact( "Unit1.Em6.ControlNodes".cm.softCam.mendrelAnodeFrontAxisZ.up.inPos )
      Contact( "Unit1.Em6.ControlNodes".cm.softCam.mendrelAnodeRearAxisY.backward.inPos )
      Contact( "Unit1.Em6.ControlNodes".cm.softCam.mendrelAnodeRearAxisZ.up.inPos )
      Coil( "Unit1.Em6.ControlNodes".stackTable."step".transition1[2220] )
   END_RUNG
   RUNG wire#w1
      Contact( "Unit1.Em6.ControlNodes".stackTable."step".transition1[2220] )
      { S7_Templates := "time_type := Time" } #statTonTime[2220].TON(pt := #delayTime, et =>)
      Move(in := #JOB_22_STEP_21, out1 => "Unit1.Em6.ControlNodes".stackTable.sequence.status.nextStep)
   END_RUNG
   // the same network as SCL:
   #_w1 := ("Unit1.Em6.ControlNodes".stackTable.sequence.status.currentStep = #JOB_22_STEP_20) AND "Unit1.Em6.ControlNodes".stackTable.sequence.status.seqActive;
   "Unit1.Em6.ControlNodes".stackTable."step".action1[2220] := #_w1 AND (NOT "Unit1.Em6.ControlNodes".cm.softCam.mendrelAnodeFrontAxisY.backward.inPos OR NOT "Unit1.Em6.ControlNodes".cm.softCam.mendrelAnodeFrontAxisZ.up.inPos OR NOT "Unit1.Em6.ControlNodes".cm.softCam.mendrelAnodeRearAxisY.backward.inPos OR NOT "Unit1.Em6.ControlNodes".cm.softCam.mendrelAnodeRearAxisZ.up.inPos);
   "Unit1.Em6.ControlNodes".stackTable."step".transition1[2220] := #_w1 AND "Unit1.Em6.ControlNodes".cm.softCam.mendrelAnodeFrontAxisY.backward.inPos AND "Unit1.Em6.ControlNodes".cm.softCam.mendrelAnodeFrontAxisZ.up.inPos AND "Unit1.Em6.ControlNodes".cm.softCam.mendrelAnodeRearAxisY.backward.inPos AND "Unit1.Em6.ControlNodes".cm.softCam.mendrelAnodeRearAxisZ.up.inPos;
   #statTonTime[2220].TON(IN := #_w1 AND "Unit1.Em6.ControlNodes".stackTable."step".transition1[2220],
                          PT := #delayTime);
   IF #statTonTime[2220].Q THEN
       "Unit1.Em6.ControlNodes".stackTable.sequence.status.nextStep := #JOB_22_STEP_21;
   END_IF;
END_REGION

REGION Network 32: Step[2221] : A.Mendrel Y,Z-Axis Work Pos
   RUNG wire#powerrail
      { S7_Templates := "SrcType := DInt" } EQ_Contact(in1 := "Unit1.Em6.ControlNodes".stackTable.sequence.status.currentStep, in2 := #JOB_22_STEP_21)
      Contact( "Unit1.Em6.ControlNodes".stackTable.sequence.status.seqActive )
      wire#w1
      I_Contact( "Unit1.Em6.ControlNodes".cm.softCam.mendrelAnodeFrontAxisY.forward.inPos )
      wire#w2
      Coil( "Unit1.Em6.ControlNodes".stackTable."step".action1[2221] )
   END_RUNG
   RUNG wire#w1
      I_Contact( "Unit1.Em6.ControlNodes".cm.softCam.mendrelAnodeFrontAxisZ.down.inPos )
   END_RUNG wire#w2
   RUNG wire#w1
      I_Contact( "Unit1.Em6.ControlNodes".cm.softCam.mendrelAnodeRearAxisY.forward.inPos )
   END_RUNG wire#w2
   RUNG wire#w1
      I_Contact( "Unit1.Em6.ControlNodes".cm.softCam.mendrelAnodeRearAxisZ.down.inPos )
   END_RUNG wire#w2
   RUNG wire#w1
      Contact( "Unit1.Em6.ControlNodes".cm.softCam.mendrelAnodeFrontAxisY.forward.inPos )
      Contact( "Unit1.Em6.ControlNodes".cm.softCam.mendrelAnodeFrontAxisZ.down.inPos )
      Contact( "Unit1.Em6.ControlNodes".cm.softCam.mendrelAnodeRearAxisY.forward.inPos )
      Contact( "Unit1.Em6.ControlNodes".cm.softCam.mendrelAnodeRearAxisZ.down.inPos )
      Coil( "Unit1.Em6.ControlNodes".stackTable."step".transition1[2221] )
   END_RUNG
   RUNG wire#w1
      Contact( "Unit1.Em6.ControlNodes".stackTable."step".transition1[2221] )
      { S7_Templates := "time_type := Time" } #statTonTime[2221].TON(pt := #delayTime, et =>)
      Move(in := #JOB_22_STEP_22, out1 => "Unit1.Em6.ControlNodes".stackTable.sequence.status.nextStep)
   END_RUNG
   // the same network as SCL:
   #_w1 := ("Unit1.Em6.ControlNodes".stackTable.sequence.status.currentStep = #JOB_22_STEP_21) AND "Unit1.Em6.ControlNodes".stackTable.sequence.status.seqActive;
   "Unit1.Em6.ControlNodes".stackTable."step".action1[2221] := #_w1 AND (NOT "Unit1.Em6.ControlNodes".cm.softCam.mendrelAnodeFrontAxisY.forward.inPos OR NOT "Unit1.Em6.ControlNodes".cm.softCam.mendrelAnodeFrontAxisZ.down.inPos OR NOT "Unit1.Em6.ControlNodes".cm.softCam.mendrelAnodeRearAxisY.forward.inPos OR NOT "Unit1.Em6.ControlNodes".cm.softCam.mendrelAnodeRearAxisZ.down.inPos);
   "Unit1.Em6.ControlNodes".stackTable."step".transition1[2221] := #_w1 AND "Unit1.Em6.ControlNodes".cm.softCam.mendrelAnodeFrontAxisY.forward.inPos AND "Unit1.Em6.ControlNodes".cm.softCam.mendrelAnodeFrontAxisZ.down.inPos AND "Unit1.Em6.ControlNodes".cm.softCam.mendrelAnodeRearAxisY.forward.inPos AND "Unit1.Em6.ControlNodes".cm.softCam.mendrelAnodeRearAxisZ.down.inPos;
   #statTonTime[2221].TON(IN := #_w1 AND "Unit1.Em6.ControlNodes".stackTable."step".transition1[2221],
                          PT := #delayTime);
   IF #statTonTime[2221].Q THEN
       "Unit1.Em6.ControlNodes".stackTable.sequence.status.nextStep := #JOB_22_STEP_22;
   END_IF;
END_REGION

REGION Network 33: Step[2222] : Stack Table → Cathode Main P&P [Clamp Done]
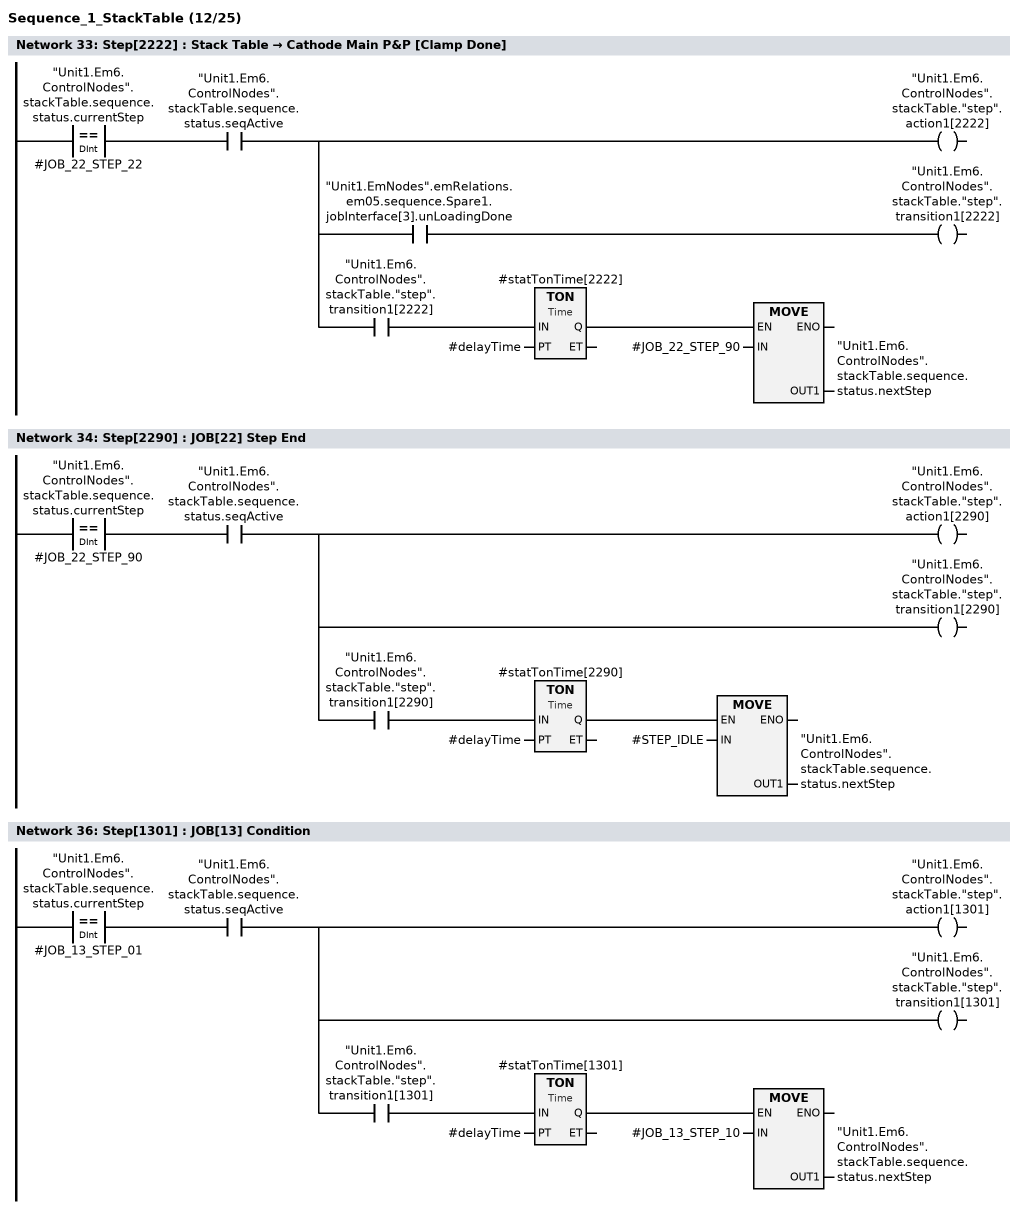
   RUNG wire#powerrail
      { S7_Templates := "SrcType := DInt" } EQ_Contact(in1 := "Unit1.Em6.ControlNodes".stackTable.sequence.status.currentStep, in2 := #JOB_22_STEP_22)
      Contact( "Unit1.Em6.ControlNodes".stackTable.sequence.status.seqActive )
      wire#w1
      Coil( "Unit1.Em6.ControlNodes".stackTable."step".action1[2222] )
   END_RUNG
   RUNG wire#w1
      Contact( "Unit1.EmNodes".emRelations.em05.sequence.Spare1.jobInterface[3].unLoadingDone )
      Coil( "Unit1.Em6.ControlNodes".stackTable."step".transition1[2222] )
   END_RUNG
   RUNG wire#w1
      Contact( "Unit1.Em6.ControlNodes".stackTable."step".transition1[2222] )
      { S7_Templates := "time_type := Time" } #statTonTime[2222].TON(pt := #delayTime, et =>)
      Move(in := #JOB_22_STEP_90, out1 => "Unit1.Em6.ControlNodes".stackTable.sequence.status.nextStep)
   END_RUNG
   // the same network as SCL:
   "Unit1.Em6.ControlNodes".stackTable."step".action1[2222] := ("Unit1.Em6.ControlNodes".stackTable.sequence.status.currentStep = #JOB_22_STEP_22) AND "Unit1.Em6.ControlNodes".stackTable.sequence.status.seqActive;
   "Unit1.Em6.ControlNodes".stackTable."step".transition1[2222] := ("Unit1.Em6.ControlNodes".stackTable.sequence.status.currentStep = #JOB_22_STEP_22) AND "Unit1.Em6.ControlNodes".stackTable.sequence.status.seqActive AND "Unit1.EmNodes".emRelations.em05.sequence.Spare1.jobInterface[3].unLoadingDone;
   #statTonTime[2222].TON(IN := ("Unit1.Em6.ControlNodes".stackTable.sequence.status.currentStep = #JOB_22_STEP_22) AND "Unit1.Em6.ControlNodes".stackTable.sequence.status.seqActive AND "Unit1.Em6.ControlNodes".stackTable."step".transition1[2222],
                          PT := #delayTime);
   IF #statTonTime[2222].Q THEN
       "Unit1.Em6.ControlNodes".stackTable.sequence.status.nextStep := #JOB_22_STEP_90;
   END_IF;
END_REGION

REGION Network 34: Step[2290] : JOB[22] Step End
   RUNG wire#powerrail
      { S7_Templates := "SrcType := DInt" } EQ_Contact(in1 := "Unit1.Em6.ControlNodes".stackTable.sequence.status.currentStep, in2 := #JOB_22_STEP_90)
      Contact( "Unit1.Em6.ControlNodes".stackTable.sequence.status.seqActive )
      wire#w1
      Coil( "Unit1.Em6.ControlNodes".stackTable."step".action1[2290] )
   END_RUNG
   RUNG wire#w1
      Coil( "Unit1.Em6.ControlNodes".stackTable."step".transition1[2290] )
   END_RUNG
   RUNG wire#w1
      Contact( "Unit1.Em6.ControlNodes".stackTable."step".transition1[2290] )
      { S7_Templates := "time_type := Time" } #statTonTime[2290].TON(pt := #delayTime, et =>)
      Move(in := #STEP_IDLE, out1 => "Unit1.Em6.ControlNodes".stackTable.sequence.status.nextStep)
   END_RUNG
   // the same network as SCL:
   "Unit1.Em6.ControlNodes".stackTable."step".action1[2290] := ("Unit1.Em6.ControlNodes".stackTable.sequence.status.currentStep = #JOB_22_STEP_90) AND "Unit1.Em6.ControlNodes".stackTable.sequence.status.seqActive;
   "Unit1.Em6.ControlNodes".stackTable."step".transition1[2290] := ("Unit1.Em6.ControlNodes".stackTable.sequence.status.currentStep = #JOB_22_STEP_90) AND "Unit1.Em6.ControlNodes".stackTable.sequence.status.seqActive;
   #statTonTime[2290].TON(IN := ("Unit1.Em6.ControlNodes".stackTable.sequence.status.currentStep = #JOB_22_STEP_90) AND "Unit1.Em6.ControlNodes".stackTable.sequence.status.seqActive AND "Unit1.Em6.ControlNodes".stackTable."step".transition1[2290],
                          PT := #delayTime);
   IF #statTonTime[2290].Q THEN
       "Unit1.Em6.ControlNodes".stackTable.sequence.status.nextStep := #STEP_IDLE;
   END_IF;
END_REGION

REGION Network 35: ******************** JOB[13] Final Roller Move [Anode → Cathode] ********************
END_REGION

REGION Network 36: Step[1301] : JOB[13] Condition
   RUNG wire#powerrail
      { S7_Templates := "SrcType := DInt" } EQ_Contact(in1 := "Unit1.Em6.ControlNodes".stackTable.sequence.status.currentStep, in2 := #JOB_13_STEP_01)
      Contact( "Unit1.Em6.ControlNodes".stackTable.sequence.status.seqActive )
      wire#w1
      Coil( "Unit1.Em6.ControlNodes".stackTable."step".action1[1301] )
   END_RUNG
   RUNG wire#w1
      Coil( "Unit1.Em6.ControlNodes".stackTable."step".transition1[1301] )
   END_RUNG
   RUNG wire#w1
      Contact( "Unit1.Em6.ControlNodes".stackTable."step".transition1[1301] )
      { S7_Templates := "time_type := Time" } #statTonTime[1301].TON(pt := #delayTime, et =>)
      Move(in := #JOB_13_STEP_10, out1 => "Unit1.Em6.ControlNodes".stackTable.sequence.status.nextStep)
   END_RUNG
   // the same network as SCL:
   "Unit1.Em6.ControlNodes".stackTable."step".action1[1301] := ("Unit1.Em6.ControlNodes".stackTable.sequence.status.currentStep = #JOB_13_STEP_01) AND "Unit1.Em6.ControlNodes".stackTable.sequence.status.seqActive;
   "Unit1.Em6.ControlNodes".stackTable."step".transition1[1301] := ("Unit1.Em6.ControlNodes".stackTable.sequence.status.currentStep = #JOB_13_STEP_01) AND "Unit1.Em6.ControlNodes".stackTable.sequence.status.seqActive;
   #statTonTime[1301].TON(IN := ("Unit1.Em6.ControlNodes".stackTable.sequence.status.currentStep = #JOB_13_STEP_01) AND "Unit1.Em6.ControlNodes".stackTable.sequence.status.seqActive AND "Unit1.Em6.ControlNodes".stackTable."step".transition1[1301],
                          PT := #delayTime);
   IF #statTonTime[1301].Q THEN
       "Unit1.Em6.ControlNodes".stackTable.sequence.status.nextStep := #JOB_13_STEP_10;
   END_IF;
END_REGION

REGION Network 37: Step[1310] : FinalRoller X-Axis Cathode Pos
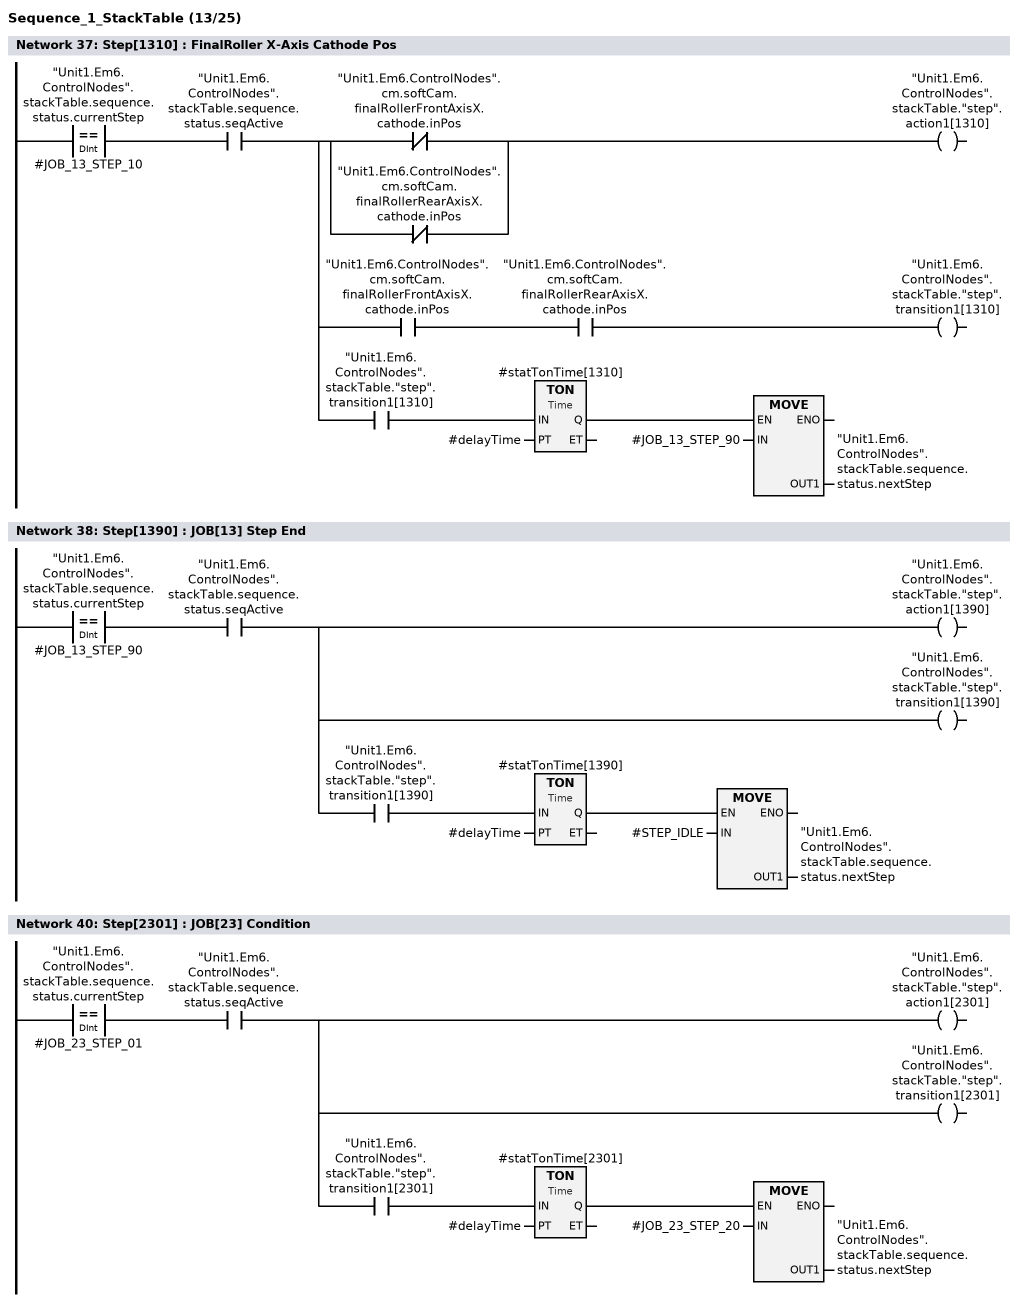
   RUNG wire#powerrail
      { S7_Templates := "SrcType := DInt" } EQ_Contact(in1 := "Unit1.Em6.ControlNodes".stackTable.sequence.status.currentStep, in2 := #JOB_13_STEP_10)
      Contact( "Unit1.Em6.ControlNodes".stackTable.sequence.status.seqActive )
      wire#w1
      I_Contact( "Unit1.Em6.ControlNodes".cm.softCam.finalRollerFrontAxisX.cathode.inPos )
      wire#w2
      Coil( "Unit1.Em6.ControlNodes".stackTable."step".action1[1310] )
   END_RUNG
   RUNG wire#w1
      I_Contact( "Unit1.Em6.ControlNodes".cm.softCam.finalRollerRearAxisX.cathode.inPos )
   END_RUNG wire#w2
   RUNG wire#w1
      Contact( "Unit1.Em6.ControlNodes".cm.softCam.finalRollerFrontAxisX.cathode.inPos )
      Contact( "Unit1.Em6.ControlNodes".cm.softCam.finalRollerRearAxisX.cathode.inPos )
      Coil( "Unit1.Em6.ControlNodes".stackTable."step".transition1[1310] )
   END_RUNG
   RUNG wire#w1
      Contact( "Unit1.Em6.ControlNodes".stackTable."step".transition1[1310] )
      { S7_Templates := "time_type := Time" } #statTonTime[1310].TON(pt := #delayTime, et =>)
      Move(in := #JOB_13_STEP_90, out1 => "Unit1.Em6.ControlNodes".stackTable.sequence.status.nextStep)
   END_RUNG
   // the same network as SCL:
   #_w1 := ("Unit1.Em6.ControlNodes".stackTable.sequence.status.currentStep = #JOB_13_STEP_10) AND "Unit1.Em6.ControlNodes".stackTable.sequence.status.seqActive;
   "Unit1.Em6.ControlNodes".stackTable."step".action1[1310] := #_w1 AND (NOT "Unit1.Em6.ControlNodes".cm.softCam.finalRollerFrontAxisX.cathode.inPos OR NOT "Unit1.Em6.ControlNodes".cm.softCam.finalRollerRearAxisX.cathode.inPos);
   "Unit1.Em6.ControlNodes".stackTable."step".transition1[1310] := #_w1 AND "Unit1.Em6.ControlNodes".cm.softCam.finalRollerFrontAxisX.cathode.inPos AND "Unit1.Em6.ControlNodes".cm.softCam.finalRollerRearAxisX.cathode.inPos;
   #statTonTime[1310].TON(IN := #_w1 AND "Unit1.Em6.ControlNodes".stackTable."step".transition1[1310],
                          PT := #delayTime);
   IF #statTonTime[1310].Q THEN
       "Unit1.Em6.ControlNodes".stackTable.sequence.status.nextStep := #JOB_13_STEP_90;
   END_IF;
END_REGION

REGION Network 38: Step[1390] : JOB[13] Step End
   RUNG wire#powerrail
      { S7_Templates := "SrcType := DInt" } EQ_Contact(in1 := "Unit1.Em6.ControlNodes".stackTable.sequence.status.currentStep, in2 := #JOB_13_STEP_90)
      Contact( "Unit1.Em6.ControlNodes".stackTable.sequence.status.seqActive )
      wire#w1
      Coil( "Unit1.Em6.ControlNodes".stackTable."step".action1[1390] )
   END_RUNG
   RUNG wire#w1
      Coil( "Unit1.Em6.ControlNodes".stackTable."step".transition1[1390] )
   END_RUNG
   RUNG wire#w1
      Contact( "Unit1.Em6.ControlNodes".stackTable."step".transition1[1390] )
      { S7_Templates := "time_type := Time" } #statTonTime[1390].TON(pt := #delayTime, et =>)
      Move(in := #STEP_IDLE, out1 => "Unit1.Em6.ControlNodes".stackTable.sequence.status.nextStep)
   END_RUNG
   // the same network as SCL:
   "Unit1.Em6.ControlNodes".stackTable."step".action1[1390] := ("Unit1.Em6.ControlNodes".stackTable.sequence.status.currentStep = #JOB_13_STEP_90) AND "Unit1.Em6.ControlNodes".stackTable.sequence.status.seqActive;
   "Unit1.Em6.ControlNodes".stackTable."step".transition1[1390] := ("Unit1.Em6.ControlNodes".stackTable.sequence.status.currentStep = #JOB_13_STEP_90) AND "Unit1.Em6.ControlNodes".stackTable.sequence.status.seqActive;
   #statTonTime[1390].TON(IN := ("Unit1.Em6.ControlNodes".stackTable.sequence.status.currentStep = #JOB_13_STEP_90) AND "Unit1.Em6.ControlNodes".stackTable.sequence.status.seqActive AND "Unit1.Em6.ControlNodes".stackTable."step".transition1[1390],
                          PT := #delayTime);
   IF #statTonTime[1390].Q THEN
       "Unit1.Em6.ControlNodes".stackTable.sequence.status.nextStep := #STEP_IDLE;
   END_IF;
END_REGION

REGION Network 39: ******************** JOB[23] Cathode Mendrel ********************
END_REGION

REGION Network 40: Step[2301] : JOB[23] Condition
   RUNG wire#powerrail
      { S7_Templates := "SrcType := DInt" } EQ_Contact(in1 := "Unit1.Em6.ControlNodes".stackTable.sequence.status.currentStep, in2 := #JOB_23_STEP_01)
      Contact( "Unit1.Em6.ControlNodes".stackTable.sequence.status.seqActive )
      wire#w1
      Coil( "Unit1.Em6.ControlNodes".stackTable."step".action1[2301] )
   END_RUNG
   RUNG wire#w1
      Coil( "Unit1.Em6.ControlNodes".stackTable."step".transition1[2301] )
   END_RUNG
   RUNG wire#w1
      Contact( "Unit1.Em6.ControlNodes".stackTable."step".transition1[2301] )
      { S7_Templates := "time_type := Time" } #statTonTime[2301].TON(pt := #delayTime, et =>)
      Move(in := #JOB_23_STEP_20, out1 => "Unit1.Em6.ControlNodes".stackTable.sequence.status.nextStep)
   END_RUNG
   // the same network as SCL:
   "Unit1.Em6.ControlNodes".stackTable."step".action1[2301] := ("Unit1.Em6.ControlNodes".stackTable.sequence.status.currentStep = #JOB_23_STEP_01) AND "Unit1.Em6.ControlNodes".stackTable.sequence.status.seqActive;
   "Unit1.Em6.ControlNodes".stackTable."step".transition1[2301] := ("Unit1.Em6.ControlNodes".stackTable.sequence.status.currentStep = #JOB_23_STEP_01) AND "Unit1.Em6.ControlNodes".stackTable.sequence.status.seqActive;
   #statTonTime[2301].TON(IN := ("Unit1.Em6.ControlNodes".stackTable.sequence.status.currentStep = #JOB_23_STEP_01) AND "Unit1.Em6.ControlNodes".stackTable.sequence.status.seqActive AND "Unit1.Em6.ControlNodes".stackTable."step".transition1[2301],
                          PT := #delayTime);
   IF #statTonTime[2301].Q THEN
       "Unit1.Em6.ControlNodes".stackTable.sequence.status.nextStep := #JOB_23_STEP_20;
   END_IF;
END_REGION

REGION Network 41: Step[2320] : C.Mendrel Y,Z-Axis Wait Pos
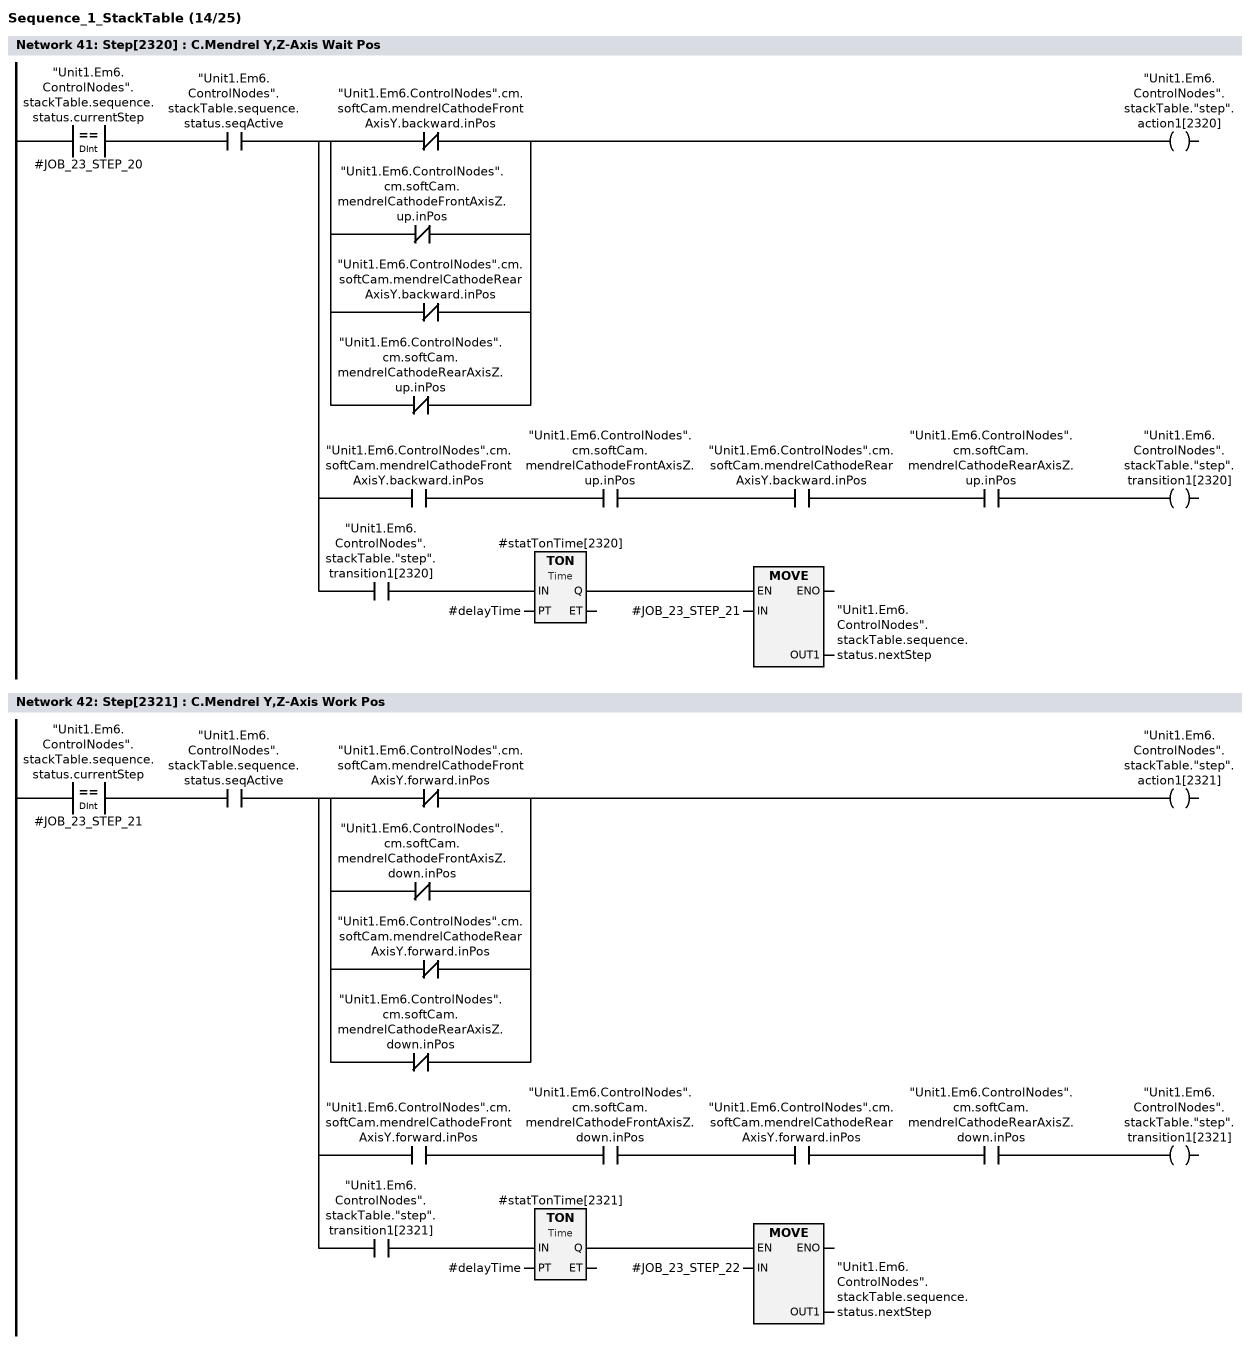
   RUNG wire#powerrail
      { S7_Templates := "SrcType := DInt" } EQ_Contact(in1 := "Unit1.Em6.ControlNodes".stackTable.sequence.status.currentStep, in2 := #JOB_23_STEP_20)
      Contact( "Unit1.Em6.ControlNodes".stackTable.sequence.status.seqActive )
      wire#w1
      I_Contact( "Unit1.Em6.ControlNodes".cm.softCam.mendrelCathodeFrontAxisY.backward.inPos )
      wire#w2
      Coil( "Unit1.Em6.ControlNodes".stackTable."step".action1[2320] )
   END_RUNG
   RUNG wire#w1
      I_Contact( "Unit1.Em6.ControlNodes".cm.softCam.mendrelCathodeFrontAxisZ.up.inPos )
   END_RUNG wire#w2
   RUNG wire#w1
      I_Contact( "Unit1.Em6.ControlNodes".cm.softCam.mendrelCathodeRearAxisY.backward.inPos )
   END_RUNG wire#w2
   RUNG wire#w1
      I_Contact( "Unit1.Em6.ControlNodes".cm.softCam.mendrelCathodeRearAxisZ.up.inPos )
   END_RUNG wire#w2
   RUNG wire#w1
      Contact( "Unit1.Em6.ControlNodes".cm.softCam.mendrelCathodeFrontAxisY.backward.inPos )
      Contact( "Unit1.Em6.ControlNodes".cm.softCam.mendrelCathodeFrontAxisZ.up.inPos )
      Contact( "Unit1.Em6.ControlNodes".cm.softCam.mendrelCathodeRearAxisY.backward.inPos )
      Contact( "Unit1.Em6.ControlNodes".cm.softCam.mendrelCathodeRearAxisZ.up.inPos )
      Coil( "Unit1.Em6.ControlNodes".stackTable."step".transition1[2320] )
   END_RUNG
   RUNG wire#w1
      Contact( "Unit1.Em6.ControlNodes".stackTable."step".transition1[2320] )
      { S7_Templates := "time_type := Time" } #statTonTime[2320].TON(pt := #delayTime, et =>)
      Move(in := #JOB_23_STEP_21, out1 => "Unit1.Em6.ControlNodes".stackTable.sequence.status.nextStep)
   END_RUNG
   // the same network as SCL:
   #_w1 := ("Unit1.Em6.ControlNodes".stackTable.sequence.status.currentStep = #JOB_23_STEP_20) AND "Unit1.Em6.ControlNodes".stackTable.sequence.status.seqActive;
   "Unit1.Em6.ControlNodes".stackTable."step".action1[2320] := #_w1 AND (NOT "Unit1.Em6.ControlNodes".cm.softCam.mendrelCathodeFrontAxisY.backward.inPos OR NOT "Unit1.Em6.ControlNodes".cm.softCam.mendrelCathodeFrontAxisZ.up.inPos OR NOT "Unit1.Em6.ControlNodes".cm.softCam.mendrelCathodeRearAxisY.backward.inPos OR NOT "Unit1.Em6.ControlNodes".cm.softCam.mendrelCathodeRearAxisZ.up.inPos);
   "Unit1.Em6.ControlNodes".stackTable."step".transition1[2320] := #_w1 AND "Unit1.Em6.ControlNodes".cm.softCam.mendrelCathodeFrontAxisY.backward.inPos AND "Unit1.Em6.ControlNodes".cm.softCam.mendrelCathodeFrontAxisZ.up.inPos AND "Unit1.Em6.ControlNodes".cm.softCam.mendrelCathodeRearAxisY.backward.inPos AND "Unit1.Em6.ControlNodes".cm.softCam.mendrelCathodeRearAxisZ.up.inPos;
   #statTonTime[2320].TON(IN := #_w1 AND "Unit1.Em6.ControlNodes".stackTable."step".transition1[2320],
                          PT := #delayTime);
   IF #statTonTime[2320].Q THEN
       "Unit1.Em6.ControlNodes".stackTable.sequence.status.nextStep := #JOB_23_STEP_21;
   END_IF;
END_REGION

REGION Network 42: Step[2321] : C.Mendrel Y,Z-Axis Work Pos
   RUNG wire#powerrail
      { S7_Templates := "SrcType := DInt" } EQ_Contact(in1 := "Unit1.Em6.ControlNodes".stackTable.sequence.status.currentStep, in2 := #JOB_23_STEP_21)
      Contact( "Unit1.Em6.ControlNodes".stackTable.sequence.status.seqActive )
      wire#w1
      I_Contact( "Unit1.Em6.ControlNodes".cm.softCam.mendrelCathodeFrontAxisY.forward.inPos )
      wire#w2
      Coil( "Unit1.Em6.ControlNodes".stackTable."step".action1[2321] )
   END_RUNG
   RUNG wire#w1
      I_Contact( "Unit1.Em6.ControlNodes".cm.softCam.mendrelCathodeFrontAxisZ.down.inPos )
   END_RUNG wire#w2
   RUNG wire#w1
      I_Contact( "Unit1.Em6.ControlNodes".cm.softCam.mendrelCathodeRearAxisY.forward.inPos )
   END_RUNG wire#w2
   RUNG wire#w1
      I_Contact( "Unit1.Em6.ControlNodes".cm.softCam.mendrelCathodeRearAxisZ.down.inPos )
   END_RUNG wire#w2
   RUNG wire#w1
      Contact( "Unit1.Em6.ControlNodes".cm.softCam.mendrelCathodeFrontAxisY.forward.inPos )
      Contact( "Unit1.Em6.ControlNodes".cm.softCam.mendrelCathodeFrontAxisZ.down.inPos )
      Contact( "Unit1.Em6.ControlNodes".cm.softCam.mendrelCathodeRearAxisY.forward.inPos )
      Contact( "Unit1.Em6.ControlNodes".cm.softCam.mendrelCathodeRearAxisZ.down.inPos )
      Coil( "Unit1.Em6.ControlNodes".stackTable."step".transition1[2321] )
   END_RUNG
   RUNG wire#w1
      Contact( "Unit1.Em6.ControlNodes".stackTable."step".transition1[2321] )
      { S7_Templates := "time_type := Time" } #statTonTime[2321].TON(pt := #delayTime, et =>)
      Move(in := #JOB_23_STEP_22, out1 => "Unit1.Em6.ControlNodes".stackTable.sequence.status.nextStep)
   END_RUNG
   // the same network as SCL:
   #_w1 := ("Unit1.Em6.ControlNodes".stackTable.sequence.status.currentStep = #JOB_23_STEP_21) AND "Unit1.Em6.ControlNodes".stackTable.sequence.status.seqActive;
   "Unit1.Em6.ControlNodes".stackTable."step".action1[2321] := #_w1 AND (NOT "Unit1.Em6.ControlNodes".cm.softCam.mendrelCathodeFrontAxisY.forward.inPos OR NOT "Unit1.Em6.ControlNodes".cm.softCam.mendrelCathodeFrontAxisZ.down.inPos OR NOT "Unit1.Em6.ControlNodes".cm.softCam.mendrelCathodeRearAxisY.forward.inPos OR NOT "Unit1.Em6.ControlNodes".cm.softCam.mendrelCathodeRearAxisZ.down.inPos);
   "Unit1.Em6.ControlNodes".stackTable."step".transition1[2321] := #_w1 AND "Unit1.Em6.ControlNodes".cm.softCam.mendrelCathodeFrontAxisY.forward.inPos AND "Unit1.Em6.ControlNodes".cm.softCam.mendrelCathodeFrontAxisZ.down.inPos AND "Unit1.Em6.ControlNodes".cm.softCam.mendrelCathodeRearAxisY.forward.inPos AND "Unit1.Em6.ControlNodes".cm.softCam.mendrelCathodeRearAxisZ.down.inPos;
   #statTonTime[2321].TON(IN := #_w1 AND "Unit1.Em6.ControlNodes".stackTable."step".transition1[2321],
                          PT := #delayTime);
   IF #statTonTime[2321].Q THEN
       "Unit1.Em6.ControlNodes".stackTable.sequence.status.nextStep := #JOB_23_STEP_22;
   END_IF;
END_REGION

REGION Network 43: Step[2322] : Stack Table → Anode Main P&P [Clamp Done]
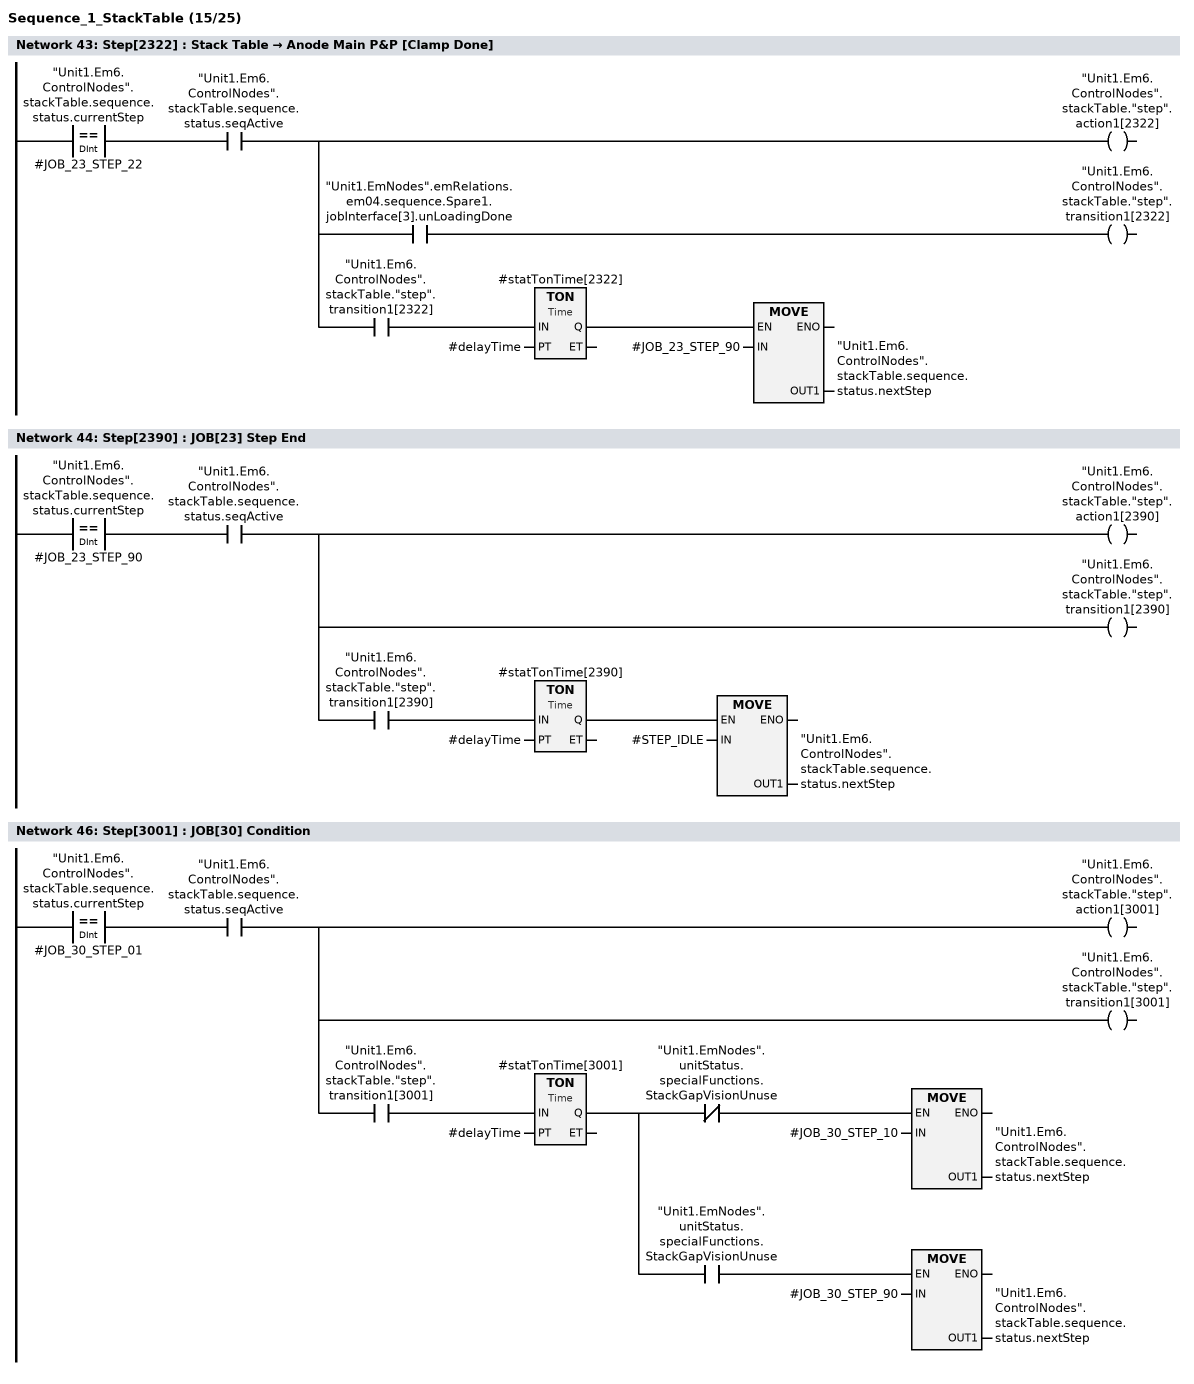
   RUNG wire#powerrail
      { S7_Templates := "SrcType := DInt" } EQ_Contact(in1 := "Unit1.Em6.ControlNodes".stackTable.sequence.status.currentStep, in2 := #JOB_23_STEP_22)
      Contact( "Unit1.Em6.ControlNodes".stackTable.sequence.status.seqActive )
      wire#w1
      Coil( "Unit1.Em6.ControlNodes".stackTable."step".action1[2322] )
   END_RUNG
   RUNG wire#w1
      Contact( "Unit1.EmNodes".emRelations.em04.sequence.Spare1.jobInterface[3].unLoadingDone )
      Coil( "Unit1.Em6.ControlNodes".stackTable."step".transition1[2322] )
   END_RUNG
   RUNG wire#w1
      Contact( "Unit1.Em6.ControlNodes".stackTable."step".transition1[2322] )
      { S7_Templates := "time_type := Time" } #statTonTime[2322].TON(pt := #delayTime, et =>)
      Move(in := #JOB_23_STEP_90, out1 => "Unit1.Em6.ControlNodes".stackTable.sequence.status.nextStep)
   END_RUNG
   // the same network as SCL:
   "Unit1.Em6.ControlNodes".stackTable."step".action1[2322] := ("Unit1.Em6.ControlNodes".stackTable.sequence.status.currentStep = #JOB_23_STEP_22) AND "Unit1.Em6.ControlNodes".stackTable.sequence.status.seqActive;
   "Unit1.Em6.ControlNodes".stackTable."step".transition1[2322] := ("Unit1.Em6.ControlNodes".stackTable.sequence.status.currentStep = #JOB_23_STEP_22) AND "Unit1.Em6.ControlNodes".stackTable.sequence.status.seqActive AND "Unit1.EmNodes".emRelations.em04.sequence.Spare1.jobInterface[3].unLoadingDone;
   #statTonTime[2322].TON(IN := ("Unit1.Em6.ControlNodes".stackTable.sequence.status.currentStep = #JOB_23_STEP_22) AND "Unit1.Em6.ControlNodes".stackTable.sequence.status.seqActive AND "Unit1.Em6.ControlNodes".stackTable."step".transition1[2322],
                          PT := #delayTime);
   IF #statTonTime[2322].Q THEN
       "Unit1.Em6.ControlNodes".stackTable.sequence.status.nextStep := #JOB_23_STEP_90;
   END_IF;
END_REGION

REGION Network 44: Step[2390] : JOB[23] Step End
   RUNG wire#powerrail
      { S7_Templates := "SrcType := DInt" } EQ_Contact(in1 := "Unit1.Em6.ControlNodes".stackTable.sequence.status.currentStep, in2 := #JOB_23_STEP_90)
      Contact( "Unit1.Em6.ControlNodes".stackTable.sequence.status.seqActive )
      wire#w1
      Coil( "Unit1.Em6.ControlNodes".stackTable."step".action1[2390] )
   END_RUNG
   RUNG wire#w1
      Coil( "Unit1.Em6.ControlNodes".stackTable."step".transition1[2390] )
   END_RUNG
   RUNG wire#w1
      Contact( "Unit1.Em6.ControlNodes".stackTable."step".transition1[2390] )
      { S7_Templates := "time_type := Time" } #statTonTime[2390].TON(pt := #delayTime, et =>)
      Move(in := #STEP_IDLE, out1 => "Unit1.Em6.ControlNodes".stackTable.sequence.status.nextStep)
   END_RUNG
   // the same network as SCL:
   "Unit1.Em6.ControlNodes".stackTable."step".action1[2390] := ("Unit1.Em6.ControlNodes".stackTable.sequence.status.currentStep = #JOB_23_STEP_90) AND "Unit1.Em6.ControlNodes".stackTable.sequence.status.seqActive;
   "Unit1.Em6.ControlNodes".stackTable."step".transition1[2390] := ("Unit1.Em6.ControlNodes".stackTable.sequence.status.currentStep = #JOB_23_STEP_90) AND "Unit1.Em6.ControlNodes".stackTable.sequence.status.seqActive;
   #statTonTime[2390].TON(IN := ("Unit1.Em6.ControlNodes".stackTable.sequence.status.currentStep = #JOB_23_STEP_90) AND "Unit1.Em6.ControlNodes".stackTable.sequence.status.seqActive AND "Unit1.Em6.ControlNodes".stackTable."step".transition1[2390],
                          PT := #delayTime);
   IF #statTonTime[2390].Q THEN
       "Unit1.Em6.ControlNodes".stackTable.sequence.status.nextStep := #STEP_IDLE;
   END_IF;
END_REGION

REGION Network 45: ******************** JOB[30] Vision ********************
END_REGION

REGION Network 46: Step[3001] : JOB[30] Condition
   RUNG wire#powerrail
      { S7_Templates := "SrcType := DInt" } EQ_Contact(in1 := "Unit1.Em6.ControlNodes".stackTable.sequence.status.currentStep, in2 := #JOB_30_STEP_01)
      Contact( "Unit1.Em6.ControlNodes".stackTable.sequence.status.seqActive )
      wire#w1
      Coil( "Unit1.Em6.ControlNodes".stackTable."step".action1[3001] )
   END_RUNG
   RUNG wire#w1
      Coil( "Unit1.Em6.ControlNodes".stackTable."step".transition1[3001] )
   END_RUNG
   RUNG wire#w1
      Contact( "Unit1.Em6.ControlNodes".stackTable."step".transition1[3001] )
      { S7_Templates := "time_type := Time" } #statTonTime[3001].TON(pt := #delayTime, et =>)
      wire#w2
      I_Contact( "Unit1.EmNodes".unitStatus.specialFunctions.StackGapVisionUnuse )
      Move(in := #JOB_30_STEP_10, out1 => "Unit1.Em6.ControlNodes".stackTable.sequence.status.nextStep)
   END_RUNG
   RUNG wire#w2
      Contact( "Unit1.EmNodes".unitStatus.specialFunctions.StackGapVisionUnuse )
      Move(in := #JOB_30_STEP_90, out1 => "Unit1.Em6.ControlNodes".stackTable.sequence.status.nextStep)
   END_RUNG
   // the same network as SCL:
   "Unit1.Em6.ControlNodes".stackTable."step".action1[3001] := ("Unit1.Em6.ControlNodes".stackTable.sequence.status.currentStep = #JOB_30_STEP_01) AND "Unit1.Em6.ControlNodes".stackTable.sequence.status.seqActive;
   "Unit1.Em6.ControlNodes".stackTable."step".transition1[3001] := ("Unit1.Em6.ControlNodes".stackTable.sequence.status.currentStep = #JOB_30_STEP_01) AND "Unit1.Em6.ControlNodes".stackTable.sequence.status.seqActive;
   #statTonTime[3001].TON(IN := ("Unit1.Em6.ControlNodes".stackTable.sequence.status.currentStep = #JOB_30_STEP_01) AND "Unit1.Em6.ControlNodes".stackTable.sequence.status.seqActive AND "Unit1.Em6.ControlNodes".stackTable."step".transition1[3001],
                          PT := #delayTime);
   IF #statTonTime[3001].Q AND NOT "Unit1.EmNodes".unitStatus.specialFunctions.StackGapVisionUnuse THEN
       "Unit1.Em6.ControlNodes".stackTable.sequence.status.nextStep := #JOB_30_STEP_10;
   END_IF;
   IF #statTonTime[3001].Q AND "Unit1.EmNodes".unitStatus.specialFunctions.StackGapVisionUnuse THEN
       "Unit1.Em6.ControlNodes".stackTable.sequence.status.nextStep := #JOB_30_STEP_90;
   END_IF;
END_REGION

REGION Network 47: Step[3010] : Vision Start
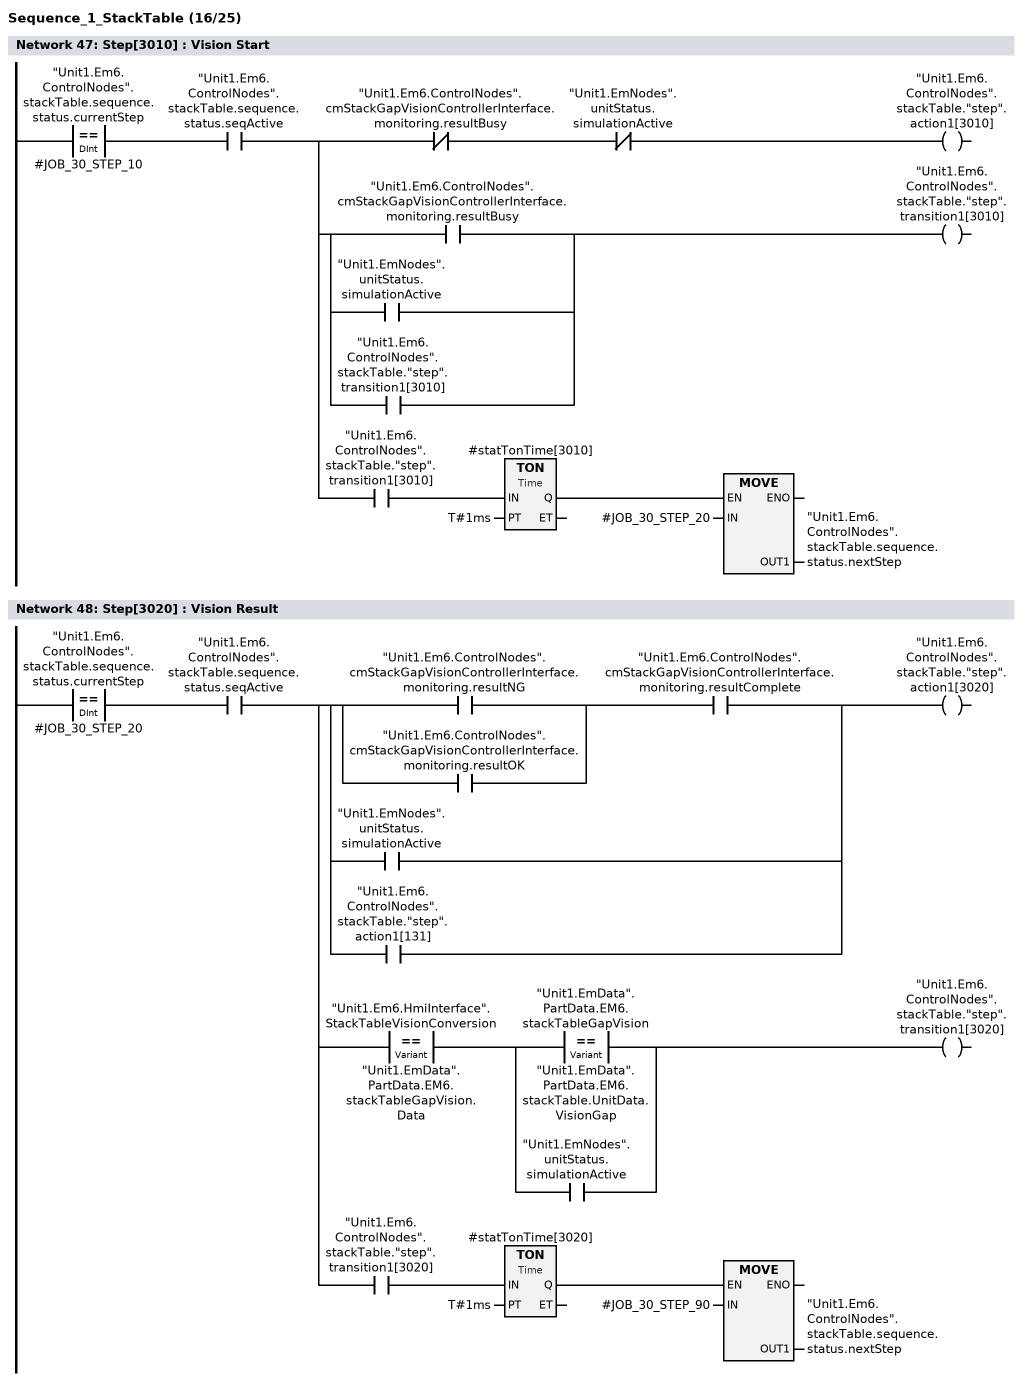
   RUNG wire#powerrail
      { S7_Templates := "SrcType := DInt" } EQ_Contact(in1 := "Unit1.Em6.ControlNodes".stackTable.sequence.status.currentStep, in2 := #JOB_30_STEP_10)
      Contact( "Unit1.Em6.ControlNodes".stackTable.sequence.status.seqActive )
      wire#w1
      I_Contact( "Unit1.Em6.ControlNodes".cmStackGapVisionControllerInterface.monitoring.resultBusy )
      I_Contact( "Unit1.EmNodes".unitStatus.simulationActive )
      Coil( "Unit1.Em6.ControlNodes".stackTable."step".action1[3010] )
   END_RUNG
   RUNG wire#w1
      Contact( "Unit1.Em6.ControlNodes".cmStackGapVisionControllerInterface.monitoring.resultBusy )
      wire#w2
      Coil( "Unit1.Em6.ControlNodes".stackTable."step".transition1[3010] )
   END_RUNG
   RUNG wire#w1
      Contact( "Unit1.EmNodes".unitStatus.simulationActive )
   END_RUNG wire#w2
   RUNG wire#w1
      Contact( "Unit1.Em6.ControlNodes".stackTable."step".transition1[3010] )
   END_RUNG wire#w2
   RUNG wire#w1
      Contact( "Unit1.Em6.ControlNodes".stackTable."step".transition1[3010] )
      { S7_Templates := "time_type := Time" } #statTonTime[3010].TON(pt := T#1ms, et =>)
      Move(in := #JOB_30_STEP_20, out1 => "Unit1.Em6.ControlNodes".stackTable.sequence.status.nextStep)
   END_RUNG
   // the same network as SCL:
   #_w1 := ("Unit1.Em6.ControlNodes".stackTable.sequence.status.currentStep = #JOB_30_STEP_10) AND "Unit1.Em6.ControlNodes".stackTable.sequence.status.seqActive;
   "Unit1.Em6.ControlNodes".stackTable."step".action1[3010] := #_w1 AND NOT "Unit1.Em6.ControlNodes".cmStackGapVisionControllerInterface.monitoring.resultBusy AND NOT "Unit1.EmNodes".unitStatus.simulationActive;
   "Unit1.Em6.ControlNodes".stackTable."step".transition1[3010] := #_w1 AND ("Unit1.Em6.ControlNodes".cmStackGapVisionControllerInterface.monitoring.resultBusy OR "Unit1.EmNodes".unitStatus.simulationActive OR "Unit1.Em6.ControlNodes".stackTable."step".transition1[3010]);
   #statTonTime[3010].TON(IN := #_w1 AND "Unit1.Em6.ControlNodes".stackTable."step".transition1[3010],
                          PT := T#1ms);
   IF #statTonTime[3010].Q THEN
       "Unit1.Em6.ControlNodes".stackTable.sequence.status.nextStep := #JOB_30_STEP_20;
   END_IF;
END_REGION

REGION Network 48: Step[3020] : Vision Result
   RUNG wire#powerrail
      { S7_Templates := "SrcType := DInt" } EQ_Contact(in1 := "Unit1.Em6.ControlNodes".stackTable.sequence.status.currentStep, in2 := #JOB_30_STEP_20)
      Contact( "Unit1.Em6.ControlNodes".stackTable.sequence.status.seqActive )
      wire#w1
      Contact( "Unit1.Em6.ControlNodes".cmStackGapVisionControllerInterface.monitoring.resultNG )
      wire#w2
      Contact( "Unit1.Em6.ControlNodes".cmStackGapVisionControllerInterface.monitoring.resultComplete )
      wire#w3
      Coil( "Unit1.Em6.ControlNodes".stackTable."step".action1[3020] )
   END_RUNG
   RUNG wire#w1
      Contact( "Unit1.Em6.ControlNodes".cmStackGapVisionControllerInterface.monitoring.resultOK )
   END_RUNG wire#w2
   RUNG wire#w1
      Contact( "Unit1.EmNodes".unitStatus.simulationActive )
   END_RUNG wire#w3
   RUNG wire#w1
      Contact( "Unit1.Em6.ControlNodes".stackTable."step".action1[131] )
   END_RUNG wire#w3
   RUNG wire#w1
      { S7_Templates := "SrcType := Variant" } EQ_Contact(in1 := "Unit1.Em6.HmiInterface".StackTableVisionConversion, in2 := "Unit1.EmData".PartData.EM6.stackTableGapVision.Data)
      wire#w4
      { S7_Templates := "SrcType := Variant" } EQ_Contact(in1 := "Unit1.EmData".PartData.EM6.stackTableGapVision, in2 := "Unit1.EmData".PartData.EM6.stackTable.UnitData.VisionGap)
      wire#w5
      Coil( "Unit1.Em6.ControlNodes".stackTable."step".transition1[3020] )
   END_RUNG
   RUNG wire#w4
      Contact( "Unit1.EmNodes".unitStatus.simulationActive )
   END_RUNG wire#w5
   RUNG wire#w1
      Contact( "Unit1.Em6.ControlNodes".stackTable."step".transition1[3020] )
      { S7_Templates := "time_type := Time" } #statTonTime[3020].TON(pt := T#1ms, et =>)
      Move(in := #JOB_30_STEP_90, out1 => "Unit1.Em6.ControlNodes".stackTable.sequence.status.nextStep)
   END_RUNG
   // the same network as SCL:
   #_w1 := ("Unit1.Em6.ControlNodes".stackTable.sequence.status.currentStep = #JOB_30_STEP_20) AND "Unit1.Em6.ControlNodes".stackTable.sequence.status.seqActive;
   "Unit1.Em6.ControlNodes".stackTable."step".action1[3020] := #_w1 AND ((("Unit1.Em6.ControlNodes".cmStackGapVisionControllerInterface.monitoring.resultNG OR "Unit1.Em6.ControlNodes".cmStackGapVisionControllerInterface.monitoring.resultOK) AND "Unit1.Em6.ControlNodes".cmStackGapVisionControllerInterface.monitoring.resultComplete) OR "Unit1.EmNodes".unitStatus.simulationActive OR "Unit1.Em6.ControlNodes".stackTable."step".action1[131]);
   "Unit1.Em6.ControlNodes".stackTable."step".transition1[3020] := #_w1 AND ("Unit1.Em6.HmiInterface".StackTableVisionConversion = "Unit1.EmData".PartData.EM6.stackTableGapVision.Data) AND (("Unit1.EmData".PartData.EM6.stackTableGapVision = "Unit1.EmData".PartData.EM6.stackTable.UnitData.VisionGap) OR "Unit1.EmNodes".unitStatus.simulationActive);
   #statTonTime[3020].TON(IN := #_w1 AND "Unit1.Em6.ControlNodes".stackTable."step".transition1[3020],
                          PT := T#1ms);
   IF #statTonTime[3020].Q THEN
       "Unit1.Em6.ControlNodes".stackTable.sequence.status.nextStep := #JOB_30_STEP_90;
   END_IF;
END_REGION

REGION Network 49: Step[3090] : JOB[30] Step End
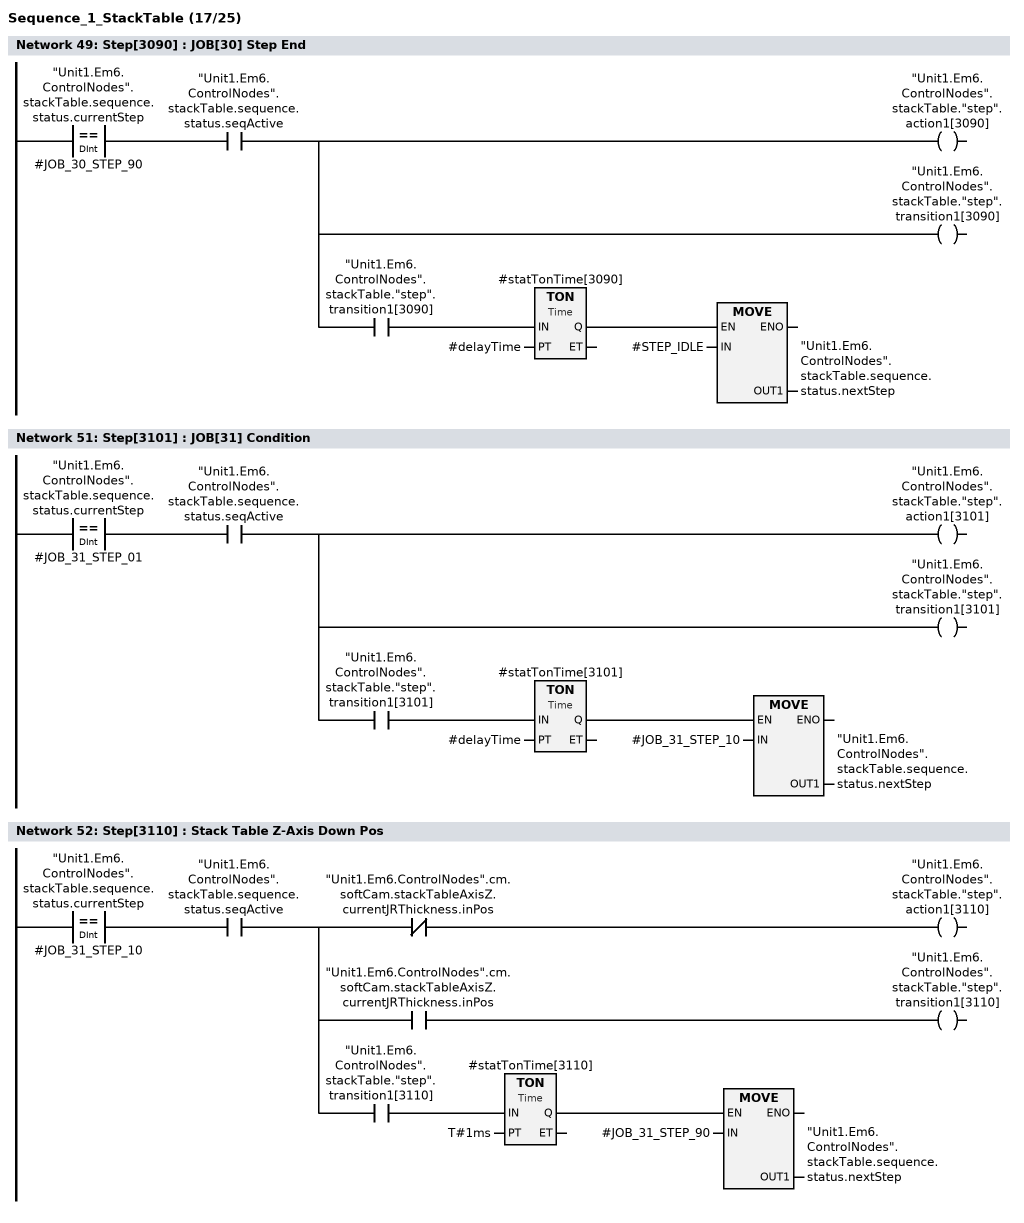
   RUNG wire#powerrail
      { S7_Templates := "SrcType := DInt" } EQ_Contact(in1 := "Unit1.Em6.ControlNodes".stackTable.sequence.status.currentStep, in2 := #JOB_30_STEP_90)
      Contact( "Unit1.Em6.ControlNodes".stackTable.sequence.status.seqActive )
      wire#w1
      Coil( "Unit1.Em6.ControlNodes".stackTable."step".action1[3090] )
   END_RUNG
   RUNG wire#w1
      Coil( "Unit1.Em6.ControlNodes".stackTable."step".transition1[3090] )
   END_RUNG
   RUNG wire#w1
      Contact( "Unit1.Em6.ControlNodes".stackTable."step".transition1[3090] )
      { S7_Templates := "time_type := Time" } #statTonTime[3090].TON(pt := #delayTime, et =>)
      Move(in := #STEP_IDLE, out1 => "Unit1.Em6.ControlNodes".stackTable.sequence.status.nextStep)
   END_RUNG
   // the same network as SCL:
   "Unit1.Em6.ControlNodes".stackTable."step".action1[3090] := ("Unit1.Em6.ControlNodes".stackTable.sequence.status.currentStep = #JOB_30_STEP_90) AND "Unit1.Em6.ControlNodes".stackTable.sequence.status.seqActive;
   "Unit1.Em6.ControlNodes".stackTable."step".transition1[3090] := ("Unit1.Em6.ControlNodes".stackTable.sequence.status.currentStep = #JOB_30_STEP_90) AND "Unit1.Em6.ControlNodes".stackTable.sequence.status.seqActive;
   #statTonTime[3090].TON(IN := ("Unit1.Em6.ControlNodes".stackTable.sequence.status.currentStep = #JOB_30_STEP_90) AND "Unit1.Em6.ControlNodes".stackTable.sequence.status.seqActive AND "Unit1.Em6.ControlNodes".stackTable."step".transition1[3090],
                          PT := #delayTime);
   IF #statTonTime[3090].Q THEN
       "Unit1.Em6.ControlNodes".stackTable.sequence.status.nextStep := #STEP_IDLE;
   END_IF;
END_REGION

REGION Network 50: ******************** JOB[31] Stack Table Down ********************
END_REGION

REGION Network 51: Step[3101] : JOB[31] Condition
   RUNG wire#powerrail
      { S7_Templates := "SrcType := DInt" } EQ_Contact(in1 := "Unit1.Em6.ControlNodes".stackTable.sequence.status.currentStep, in2 := #JOB_31_STEP_01)
      Contact( "Unit1.Em6.ControlNodes".stackTable.sequence.status.seqActive )
      wire#w1
      Coil( "Unit1.Em6.ControlNodes".stackTable."step".action1[3101] )
   END_RUNG
   RUNG wire#w1
      Coil( "Unit1.Em6.ControlNodes".stackTable."step".transition1[3101] )
   END_RUNG
   RUNG wire#w1
      Contact( "Unit1.Em6.ControlNodes".stackTable."step".transition1[3101] )
      { S7_Templates := "time_type := Time" } #statTonTime[3101].TON(pt := #delayTime, et =>)
      Move(in := #JOB_31_STEP_10, out1 => "Unit1.Em6.ControlNodes".stackTable.sequence.status.nextStep)
   END_RUNG
   // the same network as SCL:
   "Unit1.Em6.ControlNodes".stackTable."step".action1[3101] := ("Unit1.Em6.ControlNodes".stackTable.sequence.status.currentStep = #JOB_31_STEP_01) AND "Unit1.Em6.ControlNodes".stackTable.sequence.status.seqActive;
   "Unit1.Em6.ControlNodes".stackTable."step".transition1[3101] := ("Unit1.Em6.ControlNodes".stackTable.sequence.status.currentStep = #JOB_31_STEP_01) AND "Unit1.Em6.ControlNodes".stackTable.sequence.status.seqActive;
   #statTonTime[3101].TON(IN := ("Unit1.Em6.ControlNodes".stackTable.sequence.status.currentStep = #JOB_31_STEP_01) AND "Unit1.Em6.ControlNodes".stackTable.sequence.status.seqActive AND "Unit1.Em6.ControlNodes".stackTable."step".transition1[3101],
                          PT := #delayTime);
   IF #statTonTime[3101].Q THEN
       "Unit1.Em6.ControlNodes".stackTable.sequence.status.nextStep := #JOB_31_STEP_10;
   END_IF;
END_REGION

REGION Network 52: Step[3110] : Stack Table Z-Axis Down Pos
   RUNG wire#powerrail
      { S7_Templates := "SrcType := DInt" } EQ_Contact(in1 := "Unit1.Em6.ControlNodes".stackTable.sequence.status.currentStep, in2 := #JOB_31_STEP_10)
      Contact( "Unit1.Em6.ControlNodes".stackTable.sequence.status.seqActive )
      wire#w1
      I_Contact( "Unit1.Em6.ControlNodes".cm.softCam.stackTableAxisZ.currentJRThickness.inPos )
      Coil( "Unit1.Em6.ControlNodes".stackTable."step".action1[3110] )
   END_RUNG
   RUNG wire#w1
      Contact( "Unit1.Em6.ControlNodes".cm.softCam.stackTableAxisZ.currentJRThickness.inPos )
      Coil( "Unit1.Em6.ControlNodes".stackTable."step".transition1[3110] )
   END_RUNG
   RUNG wire#w1
      Contact( "Unit1.Em6.ControlNodes".stackTable."step".transition1[3110] )
      { S7_Templates := "time_type := Time" } #statTonTime[3110].TON(pt := T#1ms, et =>)
      Move(in := #JOB_31_STEP_90, out1 => "Unit1.Em6.ControlNodes".stackTable.sequence.status.nextStep)
   END_RUNG
   // the same network as SCL:
   #_w1 := ("Unit1.Em6.ControlNodes".stackTable.sequence.status.currentStep = #JOB_31_STEP_10) AND "Unit1.Em6.ControlNodes".stackTable.sequence.status.seqActive;
   "Unit1.Em6.ControlNodes".stackTable."step".action1[3110] := #_w1 AND NOT "Unit1.Em6.ControlNodes".cm.softCam.stackTableAxisZ.currentJRThickness.inPos;
   "Unit1.Em6.ControlNodes".stackTable."step".transition1[3110] := #_w1 AND "Unit1.Em6.ControlNodes".cm.softCam.stackTableAxisZ.currentJRThickness.inPos;
   #statTonTime[3110].TON(IN := #_w1 AND "Unit1.Em6.ControlNodes".stackTable."step".transition1[3110],
                          PT := T#1ms);
   IF #statTonTime[3110].Q THEN
       "Unit1.Em6.ControlNodes".stackTable.sequence.status.nextStep := #JOB_31_STEP_90;
   END_IF;
END_REGION

REGION Network 53: Step[3190] : JOB[31] Step End
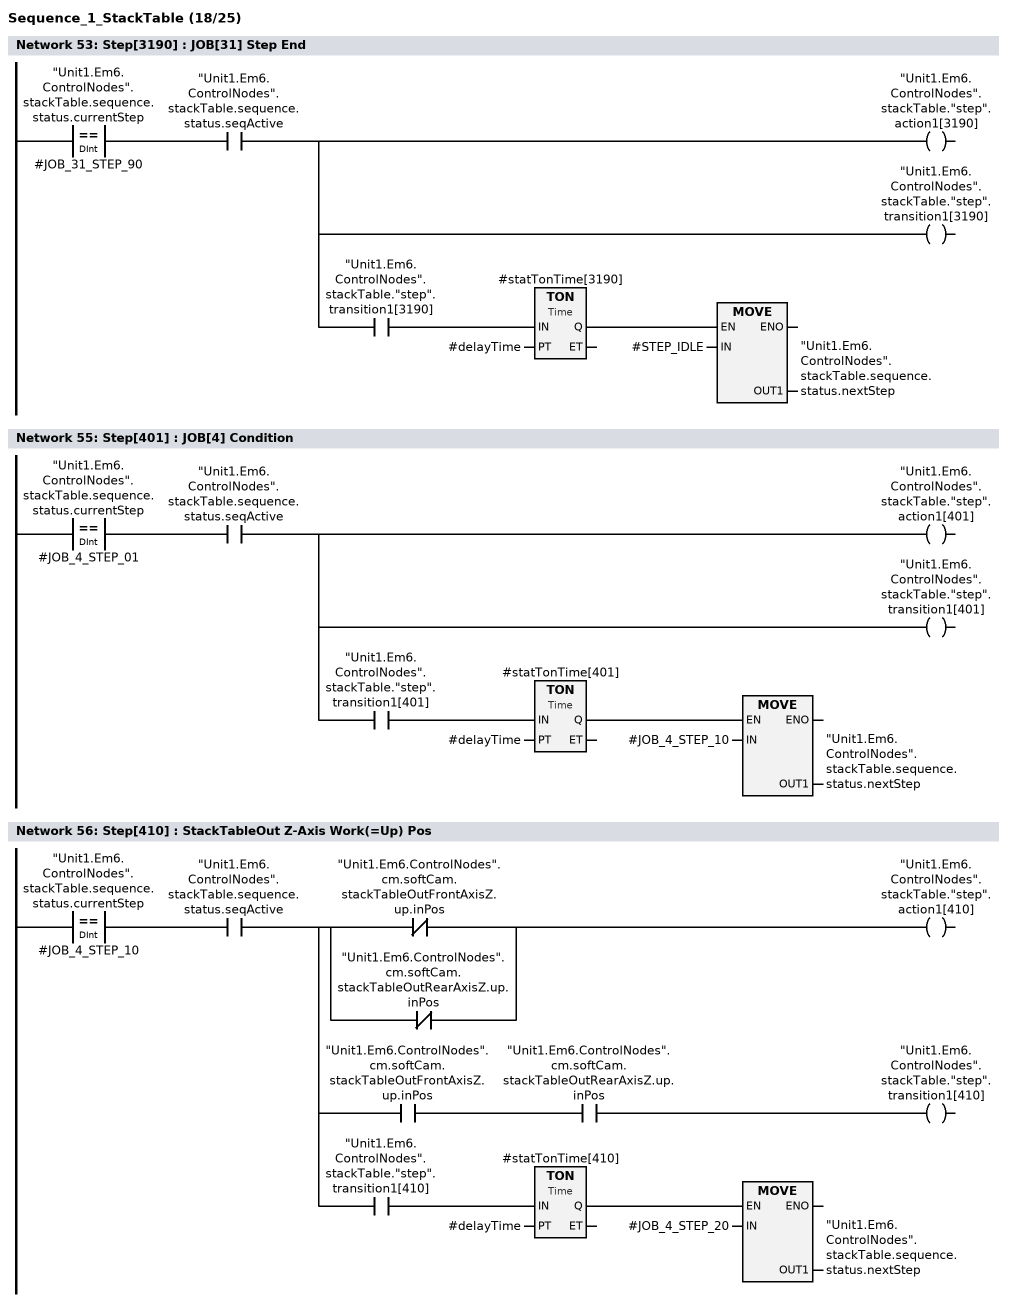
   RUNG wire#powerrail
      { S7_Templates := "SrcType := DInt" } EQ_Contact(in1 := "Unit1.Em6.ControlNodes".stackTable.sequence.status.currentStep, in2 := #JOB_31_STEP_90)
      Contact( "Unit1.Em6.ControlNodes".stackTable.sequence.status.seqActive )
      wire#w1
      Coil( "Unit1.Em6.ControlNodes".stackTable."step".action1[3190] )
   END_RUNG
   RUNG wire#w1
      Coil( "Unit1.Em6.ControlNodes".stackTable."step".transition1[3190] )
   END_RUNG
   RUNG wire#w1
      Contact( "Unit1.Em6.ControlNodes".stackTable."step".transition1[3190] )
      { S7_Templates := "time_type := Time" } #statTonTime[3190].TON(pt := #delayTime, et =>)
      Move(in := #STEP_IDLE, out1 => "Unit1.Em6.ControlNodes".stackTable.sequence.status.nextStep)
   END_RUNG
   // the same network as SCL:
   "Unit1.Em6.ControlNodes".stackTable."step".action1[3190] := ("Unit1.Em6.ControlNodes".stackTable.sequence.status.currentStep = #JOB_31_STEP_90) AND "Unit1.Em6.ControlNodes".stackTable.sequence.status.seqActive;
   "Unit1.Em6.ControlNodes".stackTable."step".transition1[3190] := ("Unit1.Em6.ControlNodes".stackTable.sequence.status.currentStep = #JOB_31_STEP_90) AND "Unit1.Em6.ControlNodes".stackTable.sequence.status.seqActive;
   #statTonTime[3190].TON(IN := ("Unit1.Em6.ControlNodes".stackTable.sequence.status.currentStep = #JOB_31_STEP_90) AND "Unit1.Em6.ControlNodes".stackTable.sequence.status.seqActive AND "Unit1.Em6.ControlNodes".stackTable."step".transition1[3190],
                          PT := #delayTime);
   IF #statTonTime[3190].Q THEN
       "Unit1.Em6.ControlNodes".stackTable.sequence.status.nextStep := #STEP_IDLE;
   END_IF;
END_REGION

REGION Network 54: *************** JOB[4] Unload ************************
END_REGION

REGION Network 55: Step[401] : JOB[4] Condition
   RUNG wire#powerrail
      { S7_Templates := "SrcType := DInt" } EQ_Contact(in1 := "Unit1.Em6.ControlNodes".stackTable.sequence.status.currentStep, in2 := #JOB_4_STEP_01)
      Contact( "Unit1.Em6.ControlNodes".stackTable.sequence.status.seqActive )
      wire#w1
      Coil( "Unit1.Em6.ControlNodes".stackTable."step".action1[401] )
   END_RUNG
   RUNG wire#w1
      Coil( "Unit1.Em6.ControlNodes".stackTable."step".transition1[401] )
   END_RUNG
   RUNG wire#w1
      Contact( "Unit1.Em6.ControlNodes".stackTable."step".transition1[401] )
      { S7_Templates := "time_type := Time" } #statTonTime[401].TON(pt := #delayTime, et =>)
      Move(in := #JOB_4_STEP_10, out1 => "Unit1.Em6.ControlNodes".stackTable.sequence.status.nextStep)
   END_RUNG
   // the same network as SCL:
   "Unit1.Em6.ControlNodes".stackTable."step".action1[401] := ("Unit1.Em6.ControlNodes".stackTable.sequence.status.currentStep = #JOB_4_STEP_01) AND "Unit1.Em6.ControlNodes".stackTable.sequence.status.seqActive;
   "Unit1.Em6.ControlNodes".stackTable."step".transition1[401] := ("Unit1.Em6.ControlNodes".stackTable.sequence.status.currentStep = #JOB_4_STEP_01) AND "Unit1.Em6.ControlNodes".stackTable.sequence.status.seqActive;
   #statTonTime[401].TON(IN := ("Unit1.Em6.ControlNodes".stackTable.sequence.status.currentStep = #JOB_4_STEP_01) AND "Unit1.Em6.ControlNodes".stackTable.sequence.status.seqActive AND "Unit1.Em6.ControlNodes".stackTable."step".transition1[401],
                         PT := #delayTime);
   IF #statTonTime[401].Q THEN
       "Unit1.Em6.ControlNodes".stackTable.sequence.status.nextStep := #JOB_4_STEP_10;
   END_IF;
END_REGION

REGION Network 56: Step[410] : StackTableOut Z-Axis Work(=Up) Pos
   RUNG wire#powerrail
      { S7_Templates := "SrcType := DInt" } EQ_Contact(in1 := "Unit1.Em6.ControlNodes".stackTable.sequence.status.currentStep, in2 := #JOB_4_STEP_10)
      Contact( "Unit1.Em6.ControlNodes".stackTable.sequence.status.seqActive )
      wire#w1
      I_Contact( "Unit1.Em6.ControlNodes".cm.softCam.stackTableOutFrontAxisZ.up.inPos )
      wire#w2
      Coil( "Unit1.Em6.ControlNodes".stackTable."step".action1[410] )
   END_RUNG
   RUNG wire#w1
      I_Contact( "Unit1.Em6.ControlNodes".cm.softCam.stackTableOutRearAxisZ.up.inPos )
   END_RUNG wire#w2
   RUNG wire#w1
      Contact( "Unit1.Em6.ControlNodes".cm.softCam.stackTableOutFrontAxisZ.up.inPos )
      Contact( "Unit1.Em6.ControlNodes".cm.softCam.stackTableOutRearAxisZ.up.inPos )
      Coil( "Unit1.Em6.ControlNodes".stackTable."step".transition1[410] )
   END_RUNG
   RUNG wire#w1
      Contact( "Unit1.Em6.ControlNodes".stackTable."step".transition1[410] )
      { S7_Templates := "time_type := Time" } #statTonTime[410].TON(pt := #delayTime, et =>)
      Move(in := #JOB_4_STEP_20, out1 => "Unit1.Em6.ControlNodes".stackTable.sequence.status.nextStep)
   END_RUNG
   // the same network as SCL:
   #_w1 := ("Unit1.Em6.ControlNodes".stackTable.sequence.status.currentStep = #JOB_4_STEP_10) AND "Unit1.Em6.ControlNodes".stackTable.sequence.status.seqActive;
   "Unit1.Em6.ControlNodes".stackTable."step".action1[410] := #_w1 AND (NOT "Unit1.Em6.ControlNodes".cm.softCam.stackTableOutFrontAxisZ.up.inPos OR NOT "Unit1.Em6.ControlNodes".cm.softCam.stackTableOutRearAxisZ.up.inPos);
   "Unit1.Em6.ControlNodes".stackTable."step".transition1[410] := #_w1 AND "Unit1.Em6.ControlNodes".cm.softCam.stackTableOutFrontAxisZ.up.inPos AND "Unit1.Em6.ControlNodes".cm.softCam.stackTableOutRearAxisZ.up.inPos;
   #statTonTime[410].TON(IN := #_w1 AND "Unit1.Em6.ControlNodes".stackTable."step".transition1[410],
                         PT := #delayTime);
   IF #statTonTime[410].Q THEN
       "Unit1.Em6.ControlNodes".stackTable.sequence.status.nextStep := #JOB_4_STEP_20;
   END_IF;
END_REGION

